# B&R Automation Studio project CControl_Gschneitner (part 7)

```iecst
		//Box 2 im Intervallbetrieb -> Dauerbetrieb u. Intervallbetrieb-Zeitfenster für alle anderen Boxen mit gleichem Lüfter sperren
		IF Box2In.IntervallbetriebEin THEN
			IF (Box2In.Ventilator1 AND Box1In.Ventilator1) OR (Box2In.Ventilator2 AND Box1In.Ventilator2) THEN
				Box1Out.DauerbetriebSperre	:= TRUE;
				FOR i := 0 TO 23 DO
					IF (Box2In.IntervallbetriebZeiten[i] = TRUE) THEN
						Box1Out.IntervallbetriebZeitenGesperrt[i]	:= TRUE;
					END_IF
				END_FOR
			END_IF
			IF (Box2In.Ventilator1 AND Box3In.Ventilator1) OR (Box2In.Ventilator2 AND Box3In.Ventilator2) THEN
				Box3Out.DauerbetriebSperre	:= TRUE;
				FOR i := 0 TO 23 DO
					IF (Box2In.IntervallbetriebZeiten[i] = TRUE) THEN
						Box3Out.IntervallbetriebZeitenGesperrt[i]	:= TRUE;
					END_IF
				END_FOR
			END_IF
			IF (Box2In.Ventilator1 AND Box4In.Ventilator1) OR (Box2In.Ventilator2 AND Box4In.Ventilator2) THEN
				Box4Out.DauerbetriebSperre	:= TRUE;
				FOR i := 0 TO 23 DO
					IF (Box2In.IntervallbetriebZeiten[i] = TRUE) THEN
						Box4Out.IntervallbetriebZeitenGesperrt[i]	:= TRUE;
					END_IF
				END_FOR
			END_IF
			IF (Box2In.Ventilator1 AND Box5In.Ventilator1) OR (Box2In.Ventilator2 AND Box5In.Ventilator2) THEN
				Box5Out.DauerbetriebSperre	:= TRUE;
				FOR i := 0 TO 23 DO
					IF (Box2In.IntervallbetriebZeiten[i] = TRUE) THEN
						Box5Out.IntervallbetriebZeitenGesperrt[i]	:= TRUE;
					END_IF
				END_FOR
			END_IF
			IF (Box2In.Ventilator1 AND Box6In.Ventilator1) OR (Box2In.Ventilator2 AND Box6In.Ventilator2) THEN
				Box6Out.DauerbetriebSperre	:= TRUE;
				FOR i := 0 TO 23 DO
					IF (Box2In.IntervallbetriebZeiten[i] = TRUE) THEN
						Box6Out.IntervallbetriebZeitenGesperrt[i]	:= TRUE;
					END_IF
				END_FOR
			END_IF
		END_IF

		//Box 3 im Intervallbetrieb -> Dauerbetrieb u. Intervallbetrieb-Zeitfenster für alle anderen Boxen mit gleichem Lüfter sperren
		IF Box3In.IntervallbetriebEin THEN
			IF (Box3In.Ventilator1 AND Box1In.Ventilator1) OR (Box3In.Ventilator2 AND Box1In.Ventilator2) THEN
				Box1Out.DauerbetriebSperre	:= TRUE;
				FOR i := 0 TO 23 DO
					IF (Box3In.IntervallbetriebZeiten[i] = TRUE) THEN
						Box1Out.IntervallbetriebZeitenGesperrt[i]	:= TRUE;
					END_IF
				END_FOR
			END_IF
			IF (Box3In.Ventilator1 AND Box2In.Ventilator1) OR (Box3In.Ventilator2 AND Box2In.Ventilator2) THEN
				Box2Out.DauerbetriebSperre	:= TRUE;
				FOR i := 0 TO 23 DO
					IF (Box3In.IntervallbetriebZeiten[i] = TRUE) THEN
						Box2Out.IntervallbetriebZeitenGesperrt[i]	:= TRUE;
					END_IF
				END_FOR
			END_IF
			IF (Box3In.Ventilator1 AND Box4In.Ventilator1) OR (Box3In.Ventilator2 AND Box4In.Ventilator2) THEN
				Box4Out.DauerbetriebSperre	:= TRUE;
				FOR i := 0 TO 23 DO
					IF (Box3In.IntervallbetriebZeiten[i] = TRUE) THEN
						Box4Out.IntervallbetriebZeitenGesperrt[i]	:= TRUE;
					END_IF
				END_FOR
			END_IF
			IF (Box3In.Ventilator1 AND Box5In.Ventilator1) OR (Box3In.Ventilator2 AND Box5In.Ventilator2) THEN
				Box5Out.DauerbetriebSperre	:= TRUE;
				FOR i := 0 TO 23 DO
					IF (Box3In.IntervallbetriebZeiten[i] = TRUE) THEN
						Box5Out.IntervallbetriebZeitenGesperrt[i]	:= TRUE;
					END_IF
				END_FOR
			END_IF
			IF (Box3In.Ventilator1 AND Box6In.Ventilator1) OR (Box3In.Ventilator2 AND Box6In.Ventilator2) THEN
				Box6Out.DauerbetriebSperre	:= TRUE;
				FOR i := 0 TO 23 DO
					IF (Box3In.IntervallbetriebZeiten[i] = TRUE) THEN
						Box6Out.IntervallbetriebZeitenGesperrt[i]	:= TRUE;
					END_IF
				END_FOR
			END_IF
		END_IF

		//Box 4 im Intervallbetrieb -> Dauerbetrieb u. Intervallbetrieb-Zeitfenster für alle anderen Boxen mit gleichem Lüfter sperren
		IF Box4In.IntervallbetriebEin THEN
			IF (Box4In.Ventilator1 AND Box1In.Ventilator1) OR (Box4In.Ventilator2 AND Box1In.Ventilator2) THEN
				Box1Out.DauerbetriebSperre	:= TRUE;
				FOR i := 0 TO 23 DO
					IF (Box4In.IntervallbetriebZeiten[i] = TRUE) THEN
						Box1Out.IntervallbetriebZeitenGesperrt[i]	:= TRUE;
					END_IF
				END_FOR
			END_IF
			IF (Box4In.Ventilator1 AND Box2In.Ventilator1) OR (Box4In.Ventilator2 AND Box2In.Ventilator2) THEN
				Box2Out.DauerbetriebSperre	:= TRUE;
				FOR i := 0 TO 23 DO
					IF (Box4In.IntervallbetriebZeiten[i] = TRUE) THEN
						Box2Out.IntervallbetriebZeitenGesperrt[i]	:= TRUE;
					END_IF
				END_FOR
			END_IF
			IF (Box4In.Ventilator1 AND Box3In.Ventilator1) OR (Box4In.Ventilator2 AND Box3In.Ventilator2) THEN
				Box3Out.DauerbetriebSperre	:= TRUE;
				FOR i := 0 TO 23 DO
					IF (Box4In.IntervallbetriebZeiten[i] = TRUE) THEN
						Box3Out.IntervallbetriebZeitenGesperrt[i]	:= TRUE;
					END_IF
				END_FOR
			END_IF
			IF (Box4In.Ventilator1 AND Box5In.Ventilator1) OR (Box4In.Ventilator2 AND Box5In.Ventilator2) THEN
				Box5Out.DauerbetriebSperre	:= TRUE;
				FOR i := 0 TO 23 DO
					IF (Box4In.IntervallbetriebZeiten[i] = TRUE) THEN
						Box5Out.IntervallbetriebZeitenGesperrt[i]	:= TRUE;
					END_IF
				END_FOR
			END_IF
			IF (Box4In.Ventilator1 AND Box6In.Ventilator1) OR (Box4In.Ventilator2 AND Box6In.Ventilator2) THEN
				Box6Out.DauerbetriebSperre	:= TRUE;
				FOR i := 0 TO 23 DO
					IF (Box4In.IntervallbetriebZeiten[i] = TRUE) THEN
						Box6Out.IntervallbetriebZeitenGesperrt[i]	:= TRUE;
					END_IF
				END_FOR
			END_IF
		END_IF

		//Box 5 im Intervallbetrieb -> Dauerbetrieb u. Intervallbetrieb-Zeitfenster für alle anderen Boxen mit gleichem Lüfter sperren
		IF Box5In.IntervallbetriebEin THEN
			IF (Box5In.Ventilator1 AND Box1In.Ventilator1) OR (Box5In.Ventilator2 AND Box1In.Ventilator2) THEN
				Box1Out.DauerbetriebSperre	:= TRUE;
				FOR i := 0 TO 23 DO
					IF (Box5In.IntervallbetriebZeiten[i] = TRUE) THEN
						Box1Out.IntervallbetriebZeitenGesperrt[i]	:= TRUE;
					END_IF
				END_FOR
			END_IF
			IF (Box5In.Ventilator1 AND Box2In.Ventilator1) OR (Box5In.Ventilator2 AND Box2In.Ventilator2) THEN
				Box2Out.DauerbetriebSperre	:= TRUE;
				FOR i := 0 TO 23 DO
					IF (Box5In.IntervallbetriebZeiten[i] = TRUE) THEN
						Box2Out.IntervallbetriebZeitenGesperrt[i]	:= TRUE;
					END_IF
				END_FOR
			END_IF
			IF (Box5In.Ventilator1 AND Box3In.Ventilator1) OR (Box5In.Ventilator2 AND Box3In.Ventilator2) THEN
				Box3Out.DauerbetriebSperre	:= TRUE;
				FOR i := 0 TO 23 DO
					IF (Box5In.IntervallbetriebZeiten[i] = TRUE) THEN
						Box3Out.IntervallbetriebZeitenGesperrt[i]	:= TRUE;
					END_IF
				END_FOR
			END_IF
			IF (Box5In.Ventilator1 AND Box4In.Ventilator1) OR (Box5In.Ventilator2 AND Box4In.Ventilator2) THEN
				Box4Out.DauerbetriebSperre	:= TRUE;
				FOR i := 0 TO 23 DO
					IF (Box5In.IntervallbetriebZeiten[i] = TRUE) THEN
						Box4Out.IntervallbetriebZeitenGesperrt[i]	:= TRUE;
					END_IF
				END_FOR
			END_IF
			IF (Box5In.Ventilator1 AND Box6In.Ventilator1) OR (Box5In.Ventilator2 AND Box6In.Ventilator2) THEN
				Box6Out.DauerbetriebSperre	:= TRUE;
				FOR i := 0 TO 23 DO
					IF (Box5In.IntervallbetriebZeiten[i] = TRUE) THEN
						Box6Out.IntervallbetriebZeitenGesperrt[i]	:= TRUE;
					END_IF
				END_FOR
			END_IF
		END_IF

		//Box 6 im Intervallbetrieb -> Dauerbetrieb u. Intervallbetrieb-Zeitfenster für alle anderen Boxen mit gleichem Lüfter sperren
		IF Box6In.IntervallbetriebEin THEN
			IF (Box6In.Ventilator1 AND Box1In.Ventilator1) OR (Box6In.Ventilator2 AND Box1In.Ventilator2) THEN
				Box1Out.DauerbetriebSperre	:= TRUE;
				FOR i := 0 TO 23 DO
					IF (Box6In.IntervallbetriebZeiten[i] = TRUE) THEN
						Box1Out.IntervallbetriebZeitenGesperrt[i]	:= TRUE;
					END_IF
				END_FOR
			END_IF
			IF (Box6In.Ventilator1 AND Box2In.Ventilator1) OR (Box6In.Ventilator2 AND Box2In.Ventilator2) THEN
				Box2Out.DauerbetriebSperre	:= TRUE;
				FOR i := 0 TO 23 DO
					IF (Box6In.IntervallbetriebZeiten[i] = TRUE) THEN
						Box2Out.IntervallbetriebZeitenGesperrt[i]	:= TRUE;
					END_IF
				END_FOR
			END_IF
			IF (Box6In.Ventilator1 AND Box3In.Ventilator1) OR (Box6In.Ventilator2 AND Box3In.Ventilator2) THEN
				Box3Out.DauerbetriebSperre	:= TRUE;
				FOR i := 0 TO 23 DO
					IF (Box6In.IntervallbetriebZeiten[i] = TRUE) THEN
						Box3Out.IntervallbetriebZeitenGesperrt[i]	:= TRUE;
					END_IF
				END_FOR
			END_IF
			IF (Box6In.Ventilator1 AND Box4In.Ventilator1) OR (Box6In.Ventilator2 AND Box4In.Ventilator2) THEN
				Box4Out.DauerbetriebSperre	:= TRUE;
				FOR i := 0 TO 23 DO
					IF (Box6In.IntervallbetriebZeiten[i] = TRUE) THEN
						Box4Out.IntervallbetriebZeitenGesperrt[i]	:= TRUE;
					END_IF
				END_FOR
			END_IF
			IF (Box6In.Ventilator1 AND Box5In.Ventilator1) OR (Box6In.Ventilator2 AND Box5In.Ventilator2) THEN
				Box5Out.DauerbetriebSperre	:= TRUE;
				FOR i := 0 TO 23 DO
					IF (Box6In.IntervallbetriebZeiten[i] = TRUE) THEN
						Box5Out.IntervallbetriebZeitenGesperrt[i]	:= TRUE;
					END_IF
				END_FOR
			END_IF
		END_IF

		//NACHTROCKNUNG AKTIVIERT =========================================================================================================================================================

		//Box 1 in der Nachtrocknung -> Nachtrocknungs-Zeitfenster für alle anderen Boxen mit gleichem Lüfter sperren
		IF Box1In.NachtrocknungEin THEN
			IF (Box1In.Ventilator1 AND Box2In.Ventilator1) OR (Box1In.Ventilator2 AND Box2In.Ventilator2) THEN
				FOR i := 0 TO 23 DO
					IF (Box1In.NachtrocknungZeiten[i] = TRUE) THEN
						Box2Out.NachtrocknungZeitenGesperrt[i]	:= TRUE;
					END_IF
				END_FOR
			END_IF
			IF (Box1In.Ventilator1 AND Box3In.Ventilator1) OR (Box1In.Ventilator2 AND Box3In.Ventilator2) THEN
				FOR i := 0 TO 23 DO
					IF (Box1In.NachtrocknungZeiten[i] = TRUE) THEN
						Box3Out.NachtrocknungZeitenGesperrt[i]	:= TRUE;
					END_IF
				END_FOR
			END_IF
			IF (Box1In.Ventilator1 AND Box4In.Ventilator1) OR (Box1In.Ventilator2 AND Box4In.Ventilator2) THEN
				FOR i := 0 TO 23 DO
					IF (Box1In.NachtrocknungZeiten[i] = TRUE) THEN
						Box4Out.NachtrocknungZeitenGesperrt[i]	:= TRUE;
					END_IF
				END_FOR
			END_IF
			IF (Box1In.Ventilator1 AND Box5In.Ventilator1) OR (Box1In.Ventilator2 AND Box5In.Ventilator2) THEN
				FOR i := 0 TO 23 DO
					IF (Box1In.NachtrocknungZeiten[i] = TRUE) THEN
						Box5Out.NachtrocknungZeitenGesperrt[i]	:= TRUE;
					END_IF
				END_FOR
			END_IF
			IF (Box1In.Ventilator1 AND Box6In.Ventilator1) OR (Box1In.Ventilator2 AND Box6In.Ventilator2) THEN
				FOR i := 0 TO 23 DO
					IF (Box1In.NachtrocknungZeiten[i] = TRUE) THEN
						Box6Out.NachtrocknungZeitenGesperrt[i]	:= TRUE;
					END_IF
				END_FOR
			END_IF
		END_IF

		//Box 2 in der Nachtrocknung -> Nachtrocknungs-Zeitfenster für alle anderen Boxen mit gleichem Lüfter sperren
		IF Box2In.NachtrocknungEin THEN
			IF (Box2In.Ventilator1 AND Box1In.Ventilator1) OR (Box2In.Ventilator2 AND Box1In.Ventilator2) THEN
				FOR i := 0 TO 23 DO
					IF (Box2In.NachtrocknungZeiten[i] = TRUE) THEN
						Box1Out.NachtrocknungZeitenGesperrt[i]	:= TRUE;
					END_IF
				END_FOR
			END_IF
			IF (Box2In.Ventilator1 AND Box3In.Ventilator1) OR (Box2In.Ventilator2 AND Box3In.Ventilator2) THEN
				FOR i := 0 TO 23 DO
					IF (Box2In.NachtrocknungZeiten[i] = TRUE) THEN
						Box3Out.NachtrocknungZeitenGesperrt[i]	:= TRUE;
					END_IF
				END_FOR
			END_IF
			IF (Box2In.Ventilator1 AND Box4In.Ventilator1) OR (Box2In.Ventilator2 AND Box4In.Ventilator2) THEN
				FOR i := 0 TO 23 DO
					IF (Box2In.NachtrocknungZeiten[i] = TRUE) THEN
						Box4Out.NachtrocknungZeitenGesperrt[i]	:= TRUE;
					END_IF
				END_FOR
			END_IF
			IF (Box2In.Ventilator1 AND Box5In.Ventilator1) OR (Box2In.Ventilator2 AND Box5In.Ventilator2) THEN
				FOR i := 0 TO 23 DO
					IF (Box2In.NachtrocknungZeiten[i] = TRUE) THEN
						Box5Out.NachtrocknungZeitenGesperrt[i]	:= TRUE;
					END_IF
				END_FOR
			END_IF
			IF (Box2In.Ventilator1 AND Box6In.Ventilator1) OR (Box2In.Ventilator2 AND Box6In.Ventilator2) THEN
				FOR i := 0 TO 23 DO
					IF (Box2In.NachtrocknungZeiten[i] = TRUE) THEN
						Box6Out.NachtrocknungZeitenGesperrt[i]	:= TRUE;
					END_IF
				END_FOR
			END_IF
		END_IF

		//Box 3 in der Nachtrocknung -> Nachtrocknungs-Zeitfenster für alle anderen Boxen mit gleichem Lüfter sperren
		IF Box3In.NachtrocknungEin THEN
			IF (Box3In.Ventilator1 AND Box1In.Ventilator1) OR (Box3In.Ventilator2 AND Box1In.Ventilator2) THEN
				FOR i := 0 TO 23 DO
					IF (Box3In.NachtrocknungZeiten[i] = TRUE) THEN
						Box1Out.NachtrocknungZeitenGesperrt[i]	:= TRUE;
					END_IF
				END_FOR
			END_IF
			IF (Box3In.Ventilator1 AND Box2In.Ventilator1) OR (Box3In.Ventilator2 AND Box2In.Ventilator2) THEN
				FOR i := 0 TO 23 DO
					IF (Box3In.NachtrocknungZeiten[i] = TRUE) THEN
						Box2Out.NachtrocknungZeitenGesperrt[i]	:= TRUE;
					END_IF
				END_FOR
			END_IF
			IF (Box3In.Ventilator1 AND Box4In.Ventilator1) OR (Box3In.Ventilator2 AND Box4In.Ventilator2) THEN
				FOR i := 0 TO 23 DO
					IF (Box3In.NachtrocknungZeiten[i] = TRUE) THEN
						Box4Out.NachtrocknungZeitenGesperrt[i]	:= TRUE;
					END_IF
				END_FOR
			END_IF
			IF (Box3In.Ventilator1 AND Box5In.Ventilator1) OR (Box3In.Ventilator2 AND Box5In.Ventilator2) THEN
				FOR i := 0 TO 23 DO
					IF (Box3In.NachtrocknungZeiten[i] = TRUE) THEN
						Box5Out.NachtrocknungZeitenGesperrt[i]	:= TRUE;
					END_IF
				END_FOR
			END_IF
			IF (Box3In.Ventilator1 AND Box6In.Ventilator1) OR (Box3In.Ventilator2 AND Box6In.Ventilator2) THEN
				FOR i := 0 TO 23 DO
					IF (Box3In.NachtrocknungZeiten[i] = TRUE) THEN
						Box6Out.NachtrocknungZeitenGesperrt[i]	:= TRUE;
					END_IF
				END_FOR
			END_IF
		END_IF

		//Box 4 in der Nachtrocknung -> Nachtrocknungs-Zeitfenster für alle anderen Boxen mit gleichem Lüfter sperren
		IF Box4In.NachtrocknungEin THEN
			IF (Box4In.Ventilator1 AND Box1In.Ventilator1) OR (Box4In.Ventilator2 AND Box1In.Ventilator2) THEN
				FOR i := 0 TO 23 DO
					IF (Box4In.NachtrocknungZeiten[i] = TRUE) THEN
						Box1Out.NachtrocknungZeitenGesperrt[i]	:= TRUE;
					END_IF
				END_FOR
			END_IF
			IF (Box4In.Ventilator1 AND Box2In.Ventilator1) OR (Box4In.Ventilator2 AND Box2In.Ventilator2) THEN
				FOR i := 0 TO 23 DO
					IF (Box4In.NachtrocknungZeiten[i] = TRUE) THEN
						Box2Out.NachtrocknungZeitenGesperrt[i]	:= TRUE;
					END_IF
				END_FOR
			END_IF
			IF (Box4In.Ventilator1 AND Box3In.Ventilator1) OR (Box4In.Ventilator2 AND Box3In.Ventilator2) THEN
				FOR i := 0 TO 23 DO
					IF (Box4In.NachtrocknungZeiten[i] = TRUE) THEN
						Box3Out.NachtrocknungZeitenGesperrt[i]	:= TRUE;
					END_IF
				END_FOR
			END_IF
			IF (Box4In.Ventilator1 AND Box5In.Ventilator1) OR (Box4In.Ventilator2 AND Box5In.Ventilator2) THEN
				FOR i := 0 TO 23 DO
					IF (Box4In.NachtrocknungZeiten[i] = TRUE) THEN
						Box5Out.NachtrocknungZeitenGesperrt[i]	:= TRUE;
					END_IF
				END_FOR
			END_IF
			IF (Box4In.Ventilator1 AND Box6In.Ventilator1) OR (Box4In.Ventilator2 AND Box6In.Ventilator2) THEN
				FOR i := 0 TO 23 DO
					IF (Box4In.NachtrocknungZeiten[i] = TRUE) THEN
						Box6Out.NachtrocknungZeitenGesperrt[i]	:= TRUE;
					END_IF
				END_FOR
			END_IF
		END_IF

		//Box 5 in der Nachtrocknung -> Nachtrocknungs-Zeitfenster für alle anderen Boxen mit gleichem Lüfter sperren
		IF Box5In.NachtrocknungEin THEN
			IF (Box5In.Ventilator1 AND Box1In.Ventilator1) OR (Box5In.Ventilator2 AND Box1In.Ventilator2) THEN
				FOR i := 0 TO 23 DO
					IF (Box5In.NachtrocknungZeiten[i] = TRUE) THEN
						Box1Out.NachtrocknungZeitenGesperrt[i]	:= TRUE;
					END_IF
				END_FOR
			END_IF
			IF (Box5In.Ventilator1 AND Box2In.Ventilator1) OR (Box5In.Ventilator2 AND Box2In.Ventilator2) THEN
				FOR i := 0 TO 23 DO
					IF (Box5In.NachtrocknungZeiten[i] = TRUE) THEN
						Box2Out.NachtrocknungZeitenGesperrt[i]	:= TRUE;
					END_IF
				END_FOR
			END_IF
			IF (Box5In.Ventilator1 AND Box3In.Ventilator1) OR (Box5In.Ventilator2 AND Box3In.Ventilator2) THEN
				FOR i := 0 TO 23 DO
					IF (Box5In.NachtrocknungZeiten[i] = TRUE) THEN
						Box3Out.NachtrocknungZeitenGesperrt[i]	:= TRUE;
					END_IF
				END_FOR
			END_IF
			IF (Box5In.Ventilator1 AND Box4In.Ventilator1) OR (Box5In.Ventilator2 AND Box4In.Ventilator2) THEN
				FOR i := 0 TO 23 DO
					IF (Box5In.NachtrocknungZeiten[i] = TRUE) THEN
						Box4Out.NachtrocknungZeitenGesperrt[i]	:= TRUE;
					END_IF
				END_FOR
			END_IF
			IF (Box5In.Ventilator1 AND Box6In.Ventilator1) OR (Box5In.Ventilator2 AND Box6In.Ventilator2) THEN
				FOR i := 0 TO 23 DO
					IF (Box5In.NachtrocknungZeiten[i] = TRUE) THEN
						Box6Out.NachtrocknungZeitenGesperrt[i]	:= TRUE;
					END_IF
				END_FOR
			END_IF
		END_IF

		//Box 6 in der Nachtrocknung -> Nachtrocknungs-Zeitfenster für alle anderen Boxen mit gleichem Lüfter sperren
		IF Box6In.NachtrocknungEin THEN
			IF (Box6In.Ventilator1 AND Box1In.Ventilator1) OR (Box6In.Ventilator2 AND Box1In.Ventilator2) THEN
				FOR i := 0 TO 23 DO
					IF (Box6In.NachtrocknungZeiten[i] = TRUE) THEN
						Box1Out.NachtrocknungZeitenGesperrt[i]	:= TRUE;
					END_IF
				END_FOR
			END_IF
			IF (Box6In.Ventilator1 AND Box2In.Ventilator1) OR (Box6In.Ventilator2 AND Box2In.Ventilator2) THEN
				FOR i := 0 TO 23 DO
					IF (Box6In.NachtrocknungZeiten[i] = TRUE) THEN
						Box2Out.NachtrocknungZeitenGesperrt[i]	:= TRUE;
					END_IF
				END_FOR
			END_IF
			IF (Box6In.Ventilator1 AND Box3In.Ventilator1) OR (Box6In.Ventilator2 AND Box3In.Ventilator2) THEN
				FOR i := 0 TO 23 DO
					IF (Box6In.NachtrocknungZeiten[i] = TRUE) THEN
						Box3Out.NachtrocknungZeitenGesperrt[i]	:= TRUE;
					END_IF
				END_FOR
			END_IF
			IF (Box6In.Ventilator1 AND Box4In.Ventilator1) OR (Box6In.Ventilator2 AND Box4In.Ventilator2) THEN
				FOR i := 0 TO 23 DO
					IF (Box6In.NachtrocknungZeiten[i] = TRUE) THEN
						Box4Out.NachtrocknungZeitenGesperrt[i]	:= TRUE;
					END_IF
				END_FOR
			END_IF
			IF (Box6In.Ventilator1 AND Box5In.Ventilator1) OR (Box6In.Ventilator2 AND Box5In.Ventilator2) THEN
				FOR i := 0 TO 23 DO
					IF (Box6In.NachtrocknungZeiten[i] = TRUE) THEN
						Box5Out.NachtrocknungZeitenGesperrt[i]	:= TRUE;
					END_IF
				END_FOR
			END_IF
		END_IF

		//Mehrere Boxen gleichzeitig belüftbar (Jalousieklappen) ******************************************************************************************************************
	ELSE

		//Box 1
		Box1Out.DauerbetriebSperre		:= FALSE;
		Box1Out.IntervallbetriebSperre	:= FALSE;
		memset(ADR(Box1Out.IntervallbetriebZeitenGesperrt), 0, SIZEOF(Box1Out.IntervallbetriebZeitenGesperrt));
		memset(ADR(Box1Out.NachtrocknungZeitenGesperrt), 0, SIZEOF(Box1Out.NachtrocknungZeitenGesperrt));

		//Box 2
		Box2Out.DauerbetriebSperre		:= FALSE;
		Box2Out.IntervallbetriebSperre	:= FALSE;
		memset(ADR(Box2Out.IntervallbetriebZeitenGesperrt), 0, SIZEOF(Box2Out.IntervallbetriebZeitenGesperrt));
		memset(ADR(Box2Out.NachtrocknungZeitenGesperrt), 0, SIZEOF(Box2Out.NachtrocknungZeitenGesperrt));

		//Box 3
		Box3Out.DauerbetriebSperre		:= FALSE;
		Box3Out.IntervallbetriebSperre	:= FALSE;
		memset(ADR(Box3Out.IntervallbetriebZeitenGesperrt), 0, SIZEOF(Box3Out.IntervallbetriebZeitenGesperrt));
		memset(ADR(Box3Out.NachtrocknungZeitenGesperrt), 0, SIZEOF(Box3Out.NachtrocknungZeitenGesperrt));

		//Box 4
		Box4Out.DauerbetriebSperre		:= FALSE;
		Box4Out.IntervallbetriebSperre	:= FALSE;
		memset(ADR(Box4Out.IntervallbetriebZeitenGesperrt), 0, SIZEOF(Box4Out.IntervallbetriebZeitenGesperrt));
		memset(ADR(Box4Out.NachtrocknungZeitenGesperrt), 0, SIZEOF(Box4Out.NachtrocknungZeitenGesperrt));

		//Box 5
		Box5Out.DauerbetriebSperre		:= FALSE;
		Box5Out.IntervallbetriebSperre	:= FALSE;
		memset(ADR(Box5Out.IntervallbetriebZeitenGesperrt), 0, SIZEOF(Box5Out.IntervallbetriebZeitenGesperrt));
		memset(ADR(Box5Out.NachtrocknungZeitenGesperrt), 0, SIZEOF(Box5Out.NachtrocknungZeitenGesperrt));

		//Box 6
		Box6Out.DauerbetriebSperre		:= FALSE;
		Box6Out.IntervallbetriebSperre	:= FALSE;
		memset(ADR(Box6Out.IntervallbetriebZeitenGesperrt), 0, SIZEOF(Box6Out.IntervallbetriebZeitenGesperrt));
		memset(ADR(Box6Out.NachtrocknungZeitenGesperrt), 0, SIZEOF(Box6Out.NachtrocknungZeitenGesperrt));

	END_IF

	//===================================================================================================================================================================================================
	//Abhängigkeiten der Boxenklappen und Bypassklappe zu den Ventilatoren ermitteln
	//(damit bei Klappenumschaltung Anlagen mit 2 Ventilatoren nur der zuständige Ventilator abgeschaltet wird)
	//===================================================================================================================================================================================================

	//Boxenklappe 1 - Ventilator 1
	Boxenkl1VonVent1Abhaengig := (Box1In.Ventilator1 AND (Box1In.StellungKlappe1 <> FBBOX_NICHT_VERWENDET)) OR
	(Box2In.Ventilator1 AND (Box2In.StellungKlappe1 <> FBBOX_NICHT_VERWENDET)) OR (Box3In.Ventilator1 AND (Box3In.StellungKlappe1 <> FBBOX_NICHT_VERWENDET)) OR
	(Box4In.Ventilator1 AND (Box4In.StellungKlappe1 <> FBBOX_NICHT_VERWENDET)) OR (Box5In.Ventilator1 AND (Box5In.StellungKlappe1 <> FBBOX_NICHT_VERWENDET)) OR
	(Box6In.Ventilator1 AND (Box6In.StellungKlappe1 <> FBBOX_NICHT_VERWENDET)) OR BoxenklVonBeidenVentAbhaengig;

	//Boxenklappe 1 - Ventilator 2
	Boxenkl1VonVent2Abhaengig := (Box1In.Ventilator2 AND (Box1In.StellungKlappe1 <> FBBOX_NICHT_VERWENDET)) OR
	(Box2In.Ventilator2 AND (Box2In.StellungKlappe1 <> FBBOX_NICHT_VERWENDET)) OR (Box3In.Ventilator2 AND (Box3In.StellungKlappe1 <> FBBOX_NICHT_VERWENDET)) OR
	(Box4In.Ventilator2 AND (Box4In.StellungKlappe1 <> FBBOX_NICHT_VERWENDET)) OR (Box5In.Ventilator2 AND (Box5In.StellungKlappe1 <> FBBOX_NICHT_VERWENDET)) OR
	(Box6In.Ventilator2 AND (Box6In.StellungKlappe1 <> FBBOX_NICHT_VERWENDET)) OR BoxenklVonBeidenVentAbhaengig;

	//Boxenklappe 2 - Ventilator 1
	Boxenkl2VonVent1Abhaengig := (Box1In.Ventilator1 AND (Box1In.StellungKlappe2 <> FBBOX_NICHT_VERWENDET)) OR
	(Box2In.Ventilator1 AND (Box2In.StellungKlappe2 <> FBBOX_NICHT_VERWENDET)) OR (Box3In.Ventilator1 AND (Box3In.StellungKlappe2 <> FBBOX_NICHT_VERWENDET)) OR
	(Box4In.Ventilator1 AND (Box4In.StellungKlappe2 <> FBBOX_NICHT_VERWENDET)) OR (Box5In.Ventilator1 AND (Box5In.StellungKlappe2 <> FBBOX_NICHT_VERWENDET)) OR
	(Box6In.Ventilator1 AND (Box6In.StellungKlappe2 <> FBBOX_NICHT_VERWENDET)) OR BoxenklVonBeidenVentAbhaengig;

	//Boxenklappe 2 - Ventilator 2
	Boxenkl2VonVent2Abhaengig := (Box1In.Ventilator2 AND (Box1In.StellungKlappe2 <> FBBOX_NICHT_VERWENDET)) OR
	(Box2In.Ventilator2 AND (Box2In.StellungKlappe2 <> FBBOX_NICHT_VERWENDET)) OR (Box3In.Ventilator2 AND (Box3In.StellungKlappe2 <> FBBOX_NICHT_VERWENDET)) OR
	(Box4In.Ventilator2 AND (Box4In.StellungKlappe2 <> FBBOX_NICHT_VERWENDET)) OR (Box5In.Ventilator2 AND (Box5In.StellungKlappe2 <> FBBOX_NICHT_VERWENDET)) OR
	(Box6In.Ventilator2 AND (Box6In.StellungKlappe2 <> FBBOX_NICHT_VERWENDET)) OR BoxenklVonBeidenVentAbhaengig;

	//Boxenklappe 3 - Ventilator 1
	Boxenkl3VonVent1Abhaengig := (Box1In.Ventilator1 AND (Box1In.StellungKlappe3 <> FBBOX_NICHT_VERWENDET)) OR
	(Box2In.Ventilator1 AND (Box2In.StellungKlappe3 <> FBBOX_NICHT_VERWENDET)) OR (Box3In.Ventilator1 AND (Box3In.StellungKlappe3 <> FBBOX_NICHT_VERWENDET)) OR
	(Box4In.Ventilator1 AND (Box4In.StellungKlappe3 <> FBBOX_NICHT_VERWENDET)) OR (Box5In.Ventilator1 AND (Box5In.StellungKlappe3 <> FBBOX_NICHT_VERWENDET)) OR
	(Box6In.Ventilator1 AND (Box6In.StellungKlappe3 <> FBBOX_NICHT_VERWENDET)) OR BoxenklVonBeidenVentAbhaengig;

	//Boxenklappe 3 - Ventilator 2
	Boxenkl3VonVent2Abhaengig := (Box1In.Ventilator2 AND (Box1In.StellungKlappe3 <> FBBOX_NICHT_VERWENDET)) OR
	(Box2In.Ventilator2 AND (Box2In.StellungKlappe3 <> FBBOX_NICHT_VERWENDET)) OR (Box3In.Ventilator2 AND (Box3In.StellungKlappe3 <> FBBOX_NICHT_VERWENDET)) OR
	(Box4In.Ventilator2 AND (Box4In.StellungKlappe3 <> FBBOX_NICHT_VERWENDET)) OR (Box5In.Ventilator2 AND (Box5In.StellungKlappe3 <> FBBOX_NICHT_VERWENDET)) OR
	(Box6In.Ventilator2 AND (Box6In.StellungKlappe3 <> FBBOX_NICHT_VERWENDET)) OR BoxenklVonBeidenVentAbhaengig;

	//Boxenklappe 4 - Ventilator 1
	Boxenkl4VonVent1Abhaengig := (Box1In.Ventilator1 AND (Box1In.StellungKlappe4 <> FBBOX_NICHT_VERWENDET)) OR
	(Box2In.Ventilator1 AND (Box2In.StellungKlappe4 <> FBBOX_NICHT_VERWENDET)) OR (Box3In.Ventilator1 AND (Box3In.StellungKlappe4 <> FBBOX_NICHT_VERWENDET)) OR
	(Box4In.Ventilator1 AND (Box4In.StellungKlappe4 <> FBBOX_NICHT_VERWENDET)) OR (Box5In.Ventilator1 AND (Box5In.StellungKlappe4 <> FBBOX_NICHT_VERWENDET)) OR
	(Box6In.Ventilator1 AND (Box6In.StellungKlappe4 <> FBBOX_NICHT_VERWENDET)) OR BoxenklVonBeidenVentAbhaengig;

	//Boxenklappe 4 - Ventilator 2
	Boxenkl4VonVent2Abhaengig := (Box1In.Ventilator2 AND (Box1In.StellungKlappe4 <> FBBOX_NICHT_VERWENDET)) OR
	(Box2In.Ventilator2 AND (Box2In.StellungKlappe4 <> FBBOX_NICHT_VERWENDET)) OR (Box3In.Ventilator2 AND (Box3In.StellungKlappe4 <> FBBOX_NICHT_VERWENDET)) OR
	(Box4In.Ventilator2 AND (Box4In.StellungKlappe4 <> FBBOX_NICHT_VERWENDET)) OR (Box5In.Ventilator2 AND (Box5In.StellungKlappe4 <> FBBOX_NICHT_VERWENDET)) OR
	(Box6In.Ventilator2 AND (Box6In.StellungKlappe4 <> FBBOX_NICHT_VERWENDET)) OR BoxenklVonBeidenVentAbhaengig;

	//Boxenklappe 5 - Ventilator 1
	Boxenkl5VonVent1Abhaengig := (Box1In.Ventilator1 AND (Box1In.StellungKlappe5 <> FBBOX_NICHT_VERWENDET)) OR
	(Box2In.Ventilator1 AND (Box2In.StellungKlappe5 <> FBBOX_NICHT_VERWENDET)) OR (Box3In.Ventilator1 AND (Box3In.StellungKlappe5 <> FBBOX_NICHT_VERWENDET)) OR
	(Box4In.Ventilator1 AND (Box4In.StellungKlappe5 <> FBBOX_NICHT_VERWENDET)) OR (Box5In.Ventilator1 AND (Box5In.StellungKlappe5 <> FBBOX_NICHT_VERWENDET)) OR
	(Box6In.Ventilator1 AND (Box6In.StellungKlappe5 <> FBBOX_NICHT_VERWENDET)) OR BoxenklVonBeidenVentAbhaengig;

	//Boxenklappe 5 - Ventilator 2
	Boxenkl5VonVent2Abhaengig := (Box1In.Ventilator2 AND (Box1In.StellungKlappe5 <> FBBOX_NICHT_VERWENDET)) OR
	(Box2In.Ventilator2 AND (Box2In.StellungKlappe5 <> FBBOX_NICHT_VERWENDET)) OR (Box3In.Ventilator2 AND (Box3In.StellungKlappe5 <> FBBOX_NICHT_VERWENDET)) OR
	(Box4In.Ventilator2 AND (Box4In.StellungKlappe5 <> FBBOX_NICHT_VERWENDET)) OR (Box5In.Ventilator2 AND (Box5In.StellungKlappe5 <> FBBOX_NICHT_VERWENDET)) OR
	(Box6In.Ventilator2 AND (Box6In.StellungKlappe5 <> FBBOX_NICHT_VERWENDET)) OR BoxenklVonBeidenVentAbhaengig;

	//Boxenklappe 6 - Ventilator 1
	Boxenkl6VonVent1Abhaengig := (Box1In.Ventilator1 AND (Box1In.StellungKlappe6 <> FBBOX_NICHT_VERWENDET)) OR
	(Box2In.Ventilator1 AND (Box2In.StellungKlappe6 <> FBBOX_NICHT_VERWENDET)) OR (Box3In.Ventilator1 AND (Box3In.StellungKlappe6 <> FBBOX_NICHT_VERWENDET)) OR
	(Box4In.Ventilator1 AND (Box4In.StellungKlappe6 <> FBBOX_NICHT_VERWENDET)) OR (Box5In.Ventilator1 AND (Box5In.StellungKlappe6 <> FBBOX_NICHT_VERWENDET)) OR
	(Box6In.Ventilator1 AND (Box6In.StellungKlappe6 <> FBBOX_NICHT_VERWENDET)) OR BoxenklVonBeidenVentAbhaengig;

	//Boxenklappe 6 - Ventilator 2
	Boxenkl6VonVent2Abhaengig := (Box1In.Ventilator2 AND (Box1In.StellungKlappe6 <> FBBOX_NICHT_VERWENDET)) OR
	(Box2In.Ventilator2 AND (Box2In.StellungKlappe6 <> FBBOX_NICHT_VERWENDET)) OR (Box3In.Ventilator2 AND (Box3In.StellungKlappe6 <> FBBOX_NICHT_VERWENDET)) OR
	(Box4In.Ventilator2 AND (Box4In.StellungKlappe6 <> FBBOX_NICHT_VERWENDET)) OR (Box5In.Ventilator2 AND (Box5In.StellungKlappe6 <> FBBOX_NICHT_VERWENDET)) OR
	(Box6In.Ventilator2 AND (Box6In.StellungKlappe6 <> FBBOX_NICHT_VERWENDET)) OR BoxenklVonBeidenVentAbhaengig;

	//Bypassklappe & Ventilator 1
	BypassklVonVent1Abhaengig := (Box1In.Ventilator1 AND Box1In.Luftentfeuchter) OR (Box2In.Ventilator1 AND Box2In.Luftentfeuchter) OR
	(Box3In.Ventilator1 AND Box3In.Luftentfeuchter) OR (Box4In.Ventilator1 AND Box4In.Luftentfeuchter) OR
	(Box5In.Ventilator1 AND Box5In.Luftentfeuchter) OR (Box6In.Ventilator1 AND Box6In.Luftentfeuchter) OR BypassklVonBeidenVentAbhaengig;

	//Bypassklappe & Ventilator 2
	BypassklVonVent2Abhaengig := (Box1In.Ventilator2 AND Box1In.Luftentfeuchter) OR (Box2In.Ventilator2 AND Box2In.Luftentfeuchter) OR
	(Box3In.Ventilator2 AND Box3In.Luftentfeuchter) OR (Box4In.Ventilator2 AND Box4In.Luftentfeuchter) OR
	(Box5In.Ventilator2 AND Box5In.Luftentfeuchter) OR (Box6In.Ventilator2 AND Box6In.Luftentfeuchter) OR BypassklVonBeidenVentAbhaengig;

END_FUNCTION_BLOCK
```

#### fbBoxenVentKlappen.st
```iecst
(* Funktionsbaustein für Ansteuerung Ventilatoren und Klappen *)
FUNCTION_BLOCK fbBoxenVentKlappen

	IF Freigabe THEN

		//Zeitticks erzeugen
		fbLascoEUhr_0(Freigabe := TRUE);
		fbLascoZdxx_0(IN := fbLascoEUhr_0.Sekunde);
		sekTick	:= fbLascoZdxx_0.Q;

		//Abfrage, ob Umschaltung Klappen erforderlich

		loc_AenderungBypassklappe		:= ((BypassklappeOeffnen AND NOT (EndlBypassOffen OR Bypassklappe.KlappeIstOffenOut)) OR
		(BypassklappeSchliessen AND NOT (EndlBypassGeschl OR Bypassklappe.KlappeIstGeschlOut))) AND (LaufzeitBypassklappe <> 0);

		loc_AenderungUmschaltklappe1	:= ((Umschaltkl1Oeffnen AND NOT (EndlUmschaltkl1Offen OR Umschaltklappe1.KlappeIstOffenOut)) OR
		(Umschaltkl1Schliessen AND NOT (EndlUmschaltkl1Geschl OR Umschaltklappe1.KlappeIstGeschlOut))) AND (LaufzeitUmschaltklappe1 <> 0);

		loc_AenderungUmschaltklappe2	:= ((Umschaltkl2Oeffnen AND NOT (EndlUmschaltkl2Offen OR Umschaltklappe2.KlappeIstOffenOut)) OR
		(Umschaltkl2Schliessen AND NOT (EndlUmschaltkl2Geschl OR Umschaltklappe2.KlappeIstGeschlOut))) AND (LaufzeitUmschaltklappe2 <> 0);

		loc_AenderungBoxenklappe1		:= Boxenklappe1Vorhanden AND ((Boxenklappe1Oeffnen AND NOT (EndlBoxenklappe1Offen OR Boxenklappe1.KlappeIstOffenOut)) OR
		(Boxenklappe1Schliessen AND NOT (EndlBoxenklappe1Geschl OR Boxenklappe1.KlappeIstGeschlOut))) AND (LaufzeitBoxenklappe1 <> 0);

		loc_AenderungBoxenklappe2		:= Boxenklappe2Vorhanden AND ((Boxenklappe2Oeffnen AND NOT (EndlBoxenklappe2Offen OR Boxenklappe2.KlappeIstOffenOut)) OR
		(Boxenklappe2Schliessen AND NOT (EndlBoxenklappe2Geschl OR Boxenklappe2.KlappeIstGeschlOut))) AND (LaufzeitBoxenklappe2 <> 0);

		loc_AenderungBoxenklappe3		:= Boxenklappe3Vorhanden AND ((Boxenklappe3Oeffnen AND NOT (EndlBoxenklappe3Offen OR Boxenklappe3.KlappeIstOffenOut)) OR
		(Boxenklappe3Schliessen AND NOT (EndlBoxenklappe3Geschl OR Boxenklappe3.KlappeIstGeschlOut))) AND (LaufzeitBoxenklappe3 <> 0);

		loc_AenderungBoxenklappe4		:= Boxenklappe4Vorhanden AND ((Boxenklappe4Oeffnen AND NOT (EndlBoxenklappe4Offen OR Boxenklappe4.KlappeIstOffenOut)) OR
		(Boxenklappe4Schliessen AND NOT (EndlBoxenklappe4Geschl OR Boxenklappe4.KlappeIstGeschlOut))) AND (LaufzeitBoxenklappe4 <> 0);

		loc_AenderungBoxenklappe5		:= Boxenklappe5Vorhanden AND ((Boxenklappe5Oeffnen AND NOT (EndlBoxenklappe5Offen OR Boxenklappe5.KlappeIstOffenOut)) OR
		(Boxenklappe5Schliessen AND NOT (EndlBoxenklappe5Geschl OR Boxenklappe5.KlappeIstGeschlOut))) AND (LaufzeitBoxenklappe5 <> 0);

		loc_AenderungBoxenklappe6		:= Boxenklappe6Vorhanden AND ((Boxenklappe6Oeffnen AND NOT (EndlBoxenklappe6Offen OR Boxenklappe6.KlappeIstOffenOut)) OR
		(Boxenklappe6Schliessen AND NOT (EndlBoxenklappe6Geschl OR Boxenklappe6.KlappeIstGeschlOut))) AND (LaufzeitBoxenklappe6 <> 0);

		//Umschaltung erforderlich bei Ventilator 1
		loc_UmschaltungErforderlVent1		:= (loc_AenderungBypassklappe AND BypassklVonVent1Abhaengig) OR
		(loc_AenderungUmschaltklappe1 AND UmluftklVonVent1Abhaengig) OR (loc_AenderungUmschaltklappe2 AND UmluftklVonVent1Abhaengig) OR
		(loc_AenderungBoxenklappe1 AND Boxenkl1VonVent1Abhaengig) OR (loc_AenderungBoxenklappe2 AND Boxenkl2VonVent1Abhaengig) OR
		(loc_AenderungBoxenklappe3 AND Boxenkl3VonVent1Abhaengig) OR (loc_AenderungBoxenklappe4 AND Boxenkl4VonVent1Abhaengig) OR
		(loc_AenderungBoxenklappe5 AND Boxenkl5VonVent1Abhaengig) OR (loc_AenderungBoxenklappe6 AND Boxenkl6VonVent1Abhaengig);

		//Umschaltung erfoderlich bei Ventilator 2
		loc_UmschaltungErforderlVent2		:= (loc_AenderungBypassklappe AND BypassklVonVent2Abhaengig) OR
		(loc_AenderungUmschaltklappe1 AND UmluftklVonVent2Abhaengig) OR (loc_AenderungUmschaltklappe2 AND UmluftklVonVent2Abhaengig) OR
		(loc_AenderungBoxenklappe1 AND Boxenkl1VonVent2Abhaengig) OR (loc_AenderungBoxenklappe2 AND Boxenkl2VonVent2Abhaengig) OR
		(loc_AenderungBoxenklappe3 AND Boxenkl3VonVent2Abhaengig) OR (loc_AenderungBoxenklappe4 AND Boxenkl4VonVent2Abhaengig) OR
		(loc_AenderungBoxenklappe5 AND Boxenkl5VonVent2Abhaengig) OR (loc_AenderungBoxenklappe6 AND Boxenkl6VonVent2Abhaengig);

		//Funktionsbaustein Ansteuerung FU Ventilator 1
		fbFuVentilator1.AnsprechZeitFU		:= 5;
		fbFuVentilator1.BetrMldg			:= Ventilator1InBetrieb;
		fbFuVentilator1.MinDrehzahl			:= DrehzahlVent1Min;
		fbFuVentilator1.MaxDrehzahl			:= DrehzahlVent1Max;
		fbFuVentilator1.RampeUpSek			:= RampeVent1Up;
		fbFuVentilator1.RampeDownSek		:= RampeVent1Down;
		fbFuVentilator1.Reset				:= QuitFehler;
		fbFuVentilator1.Tick				:= sekTick;
		fbFuVentilator1();
		FreigabeVentilator1Out				:= fbFuVentilator1.BetriebFU;
		DrehzahlVent1Out					:= fbFuVentilator1.DrehzahlFU;
		FehlerFuVentilator1					:= fbFuVentilator1.StoerungFU;

		//Funktionsbaustein Ansteuerung FU Ventilator 2
		fbFuVentilator2.AnsprechZeitFU		:= 5;
		fbFuVentilator2.BetrMldg			:= Ventilator2InBetrieb;
		fbFuVentilator2.MinDrehzahl			:= DrehzahlVent2Min;
		fbFuVentilator2.MaxDrehzahl			:= DrehzahlVent2Max;
		fbFuVentilator2.RampeUpSek			:= RampeVent2Up;
		fbFuVentilator2.RampeDownSek		:= RampeVent2Down;
		fbFuVentilator2.Reset				:= QuitFehler;
		fbFuVentilator2.Tick				:= sekTick;
		fbFuVentilator2();
		FreigabeVentilator2Out				:= fbFuVentilator2.BetriebFU;
		DrehzahlVent2Out					:= fbFuVentilator2.DrehzahlFU;
		FehlerFuVentilator2					:= fbFuVentilator2.StoerungFU;

		//Funktionsbausteine Klappen
		Bypassklappe.EndlagenVhd			:= EndlagenVhdBypassklappe;
		Bypassklappe.EndlageOffen			:= EndlBypassOffen;
		Bypassklappe.EndlageGeschl			:= EndlBypassGeschl;
		Bypassklappe.LaufzeitOeffnen		:= LaufzeitBypassklappe;
		Bypassklappe.LaufzeitSchliessen		:= LaufzeitBypassklappe;
		Bypassklappe.Stoerung				:= EndlBypassGeschl AND EndlBypassOffen;
		Bypassklappe.QuitFehler				:= QuitFehler;
		Bypassklappe();
		BypassOeffnenOut					:= Bypassklappe.OeffnenOut;
		BypassSchliessenOut					:= Bypassklappe.SchliessenOut;
		FehlerLaufzeitBypass				:= Bypassklappe.FehlerLaufzeitOeffnen OR Bypassklappe.FehlerLaufzeitSchliessen;
		BypassklappeIstGeschl				:= Bypassklappe.KlappeIstGeschlOut;
		BypassklappeIstOffen				:= Bypassklappe.KlappeIstOffenOut;

		Umschaltklappe1.EndlagenVhd			:= EndlagenVhdUmschaltklappe1;
		Umschaltklappe1.EndlageOffen		:= EndlUmschaltkl1Offen;
		Umschaltklappe1.EndlageGeschl		:= EndlUmschaltkl1Geschl;
		Umschaltklappe1.LaufzeitOeffnen		:= LaufzeitUmschaltklappe1;
		Umschaltklappe1.LaufzeitSchliessen	:= LaufzeitUmschaltklappe1;
		Umschaltklappe1.Stoerung			:= EndlUmschaltkl1Offen AND EndlUmschaltkl1Geschl;
		Umschaltklappe1.QuitFehler			:= QuitFehler;
		Umschaltklappe1();
		Umschaltkl1OeffnenOut				:= Umschaltklappe1.OeffnenOut;
		Umschaltkl1SchliessenOut			:= Umschaltklappe1.SchliessenOut;
		FehlerLaufzeitUmschaltkl1			:= Umschaltklappe1.FehlerLaufzeitOeffnen OR Umschaltklappe1.FehlerLaufzeitSchliessen;
		Umschaltklappe1IstGeschl			:= Umschaltklappe1.KlappeIstGeschlOut;
		Umschaltklappe1IstOffen				:= Umschaltklappe1.KlappeIstOffenOut;

		Umschaltklappe2.EndlagenVhd			:= EndlagenVhdUmschaltklappe2;
		Umschaltklappe2.EndlageOffen		:= EndlUmschaltkl2Offen;
		Umschaltklappe2.EndlageGeschl		:= EndlUmschaltkl2Geschl;
		Umschaltklappe2.LaufzeitOeffnen		:= LaufzeitUmschaltklappe2;
		Umschaltklappe2.LaufzeitSchliessen	:= LaufzeitUmschaltklappe2;
		Umschaltklappe2.Stoerung			:= EndlUmschaltkl2Offen AND EndlUmschaltkl2Geschl;
		Umschaltklappe2.QuitFehler			:= QuitFehler;
		Umschaltklappe2();
		Umschaltkl2OeffnenOut				:= Umschaltklappe2.OeffnenOut;
		Umschaltkl2SchliessenOut			:= Umschaltklappe2.SchliessenOut;
		FehlerLaufzeitUmschaltkl2			:= Umschaltklappe2.FehlerLaufzeitOeffnen OR Umschaltklappe2.FehlerLaufzeitSchliessen;
		Umschaltklappe2IstGeschl			:= Umschaltklappe2.KlappeIstGeschlOut;
		Umschaltklappe2IstOffen				:= Umschaltklappe2.KlappeIstOffenOut;

		Boxenklappe1.EndlagenVhd			:= EndlagenVhdBoxenklappe1;
		Boxenklappe1.EndlageOffen			:= EndlBoxenklappe1Offen;
		Boxenklappe1.EndlageGeschl			:= EndlBoxenklappe1Geschl;
		Boxenklappe1.LaufzeitOeffnen		:= LaufzeitBoxenklappe1;
		Boxenklappe1.LaufzeitSchliessen		:= LaufzeitBoxenklappe1;
		Boxenklappe1.Stoerung				:= EndlBoxenklappe1Offen AND EndlBoxenklappe1Geschl;
		Boxenklappe1.QuitFehler				:= QuitFehler;
		Boxenklappe1();
		Boxenklappe1IstGeschl				:= Boxenklappe1.KlappeIstGeschlOut;
		Boxenklappe1IstOffen				:= Boxenklappe1.KlappeIstOffenOut;
		IF Boxenklappe1Vorhanden THEN
			Boxenklappe1OeffnenOut				:= Boxenklappe1.OeffnenOut;
			Boxenklappe1SchliessenOut			:= Boxenklappe1.SchliessenOut;
			FehlerLaufzeitKlappeBox1			:= Boxenklappe1.FehlerLaufzeitOeffnen OR Boxenklappe1.FehlerLaufzeitSchliessen;
		ELSE
			Boxenklappe1OeffnenOut				:= FALSE;
			Boxenklappe1SchliessenOut			:= FALSE;
			FehlerLaufzeitKlappeBox1			:= FALSE;
		END_IF

		Boxenklappe2.EndlagenVhd			:= EndlagenVhdBoxenklappe2;
		Boxenklappe2.EndlageOffen			:= EndlBoxenklappe2Offen;
		Boxenklappe2.EndlageGeschl			:= EndlBoxenklappe2Geschl;
		Boxenklappe2.LaufzeitOeffnen		:= LaufzeitBoxenklappe2;
		Boxenklappe2.LaufzeitSchliessen		:= LaufzeitBoxenklappe2;
		Boxenklappe2.Stoerung				:= EndlBoxenklappe2Offen AND EndlBoxenklappe2Geschl;
		Boxenklappe2.QuitFehler				:= QuitFehler;
		Boxenklappe2();
		Boxenklappe2IstGeschl				:= Boxenklappe2.KlappeIstGeschlOut;
		Boxenklappe2IstOffen				:= Boxenklappe2.KlappeIstOffenOut;
		IF Boxenklappe2Vorhanden THEN
			Boxenklappe2OeffnenOut				:= Boxenklappe2.OeffnenOut;
			Boxenklappe2SchliessenOut			:= Boxenklappe2.SchliessenOut;
			FehlerLaufzeitKlappeBox2			:= Boxenklappe2.FehlerLaufzeitOeffnen OR Boxenklappe2.FehlerLaufzeitSchliessen;
		ELSE
			Boxenklappe2OeffnenOut				:= FALSE;
			Boxenklappe2SchliessenOut			:= FALSE;
			FehlerLaufzeitKlappeBox2			:= FALSE;
		END_IF

		Boxenklappe3.EndlagenVhd			:= EndlagenVhdBoxenklappe3;
		Boxenklappe3.EndlageOffen			:= EndlBoxenklappe3Offen;
		Boxenklappe3.EndlageGeschl			:= EndlBoxenklappe3Geschl;
		Boxenklappe3.LaufzeitOeffnen		:= LaufzeitBoxenklappe3;
		Boxenklappe3.LaufzeitSchliessen		:= LaufzeitBoxenklappe3;
		Boxenklappe3.Stoerung				:= EndlBoxenklappe3Offen AND EndlBoxenklappe3Geschl;
		Boxenklappe3.QuitFehler				:= QuitFehler;
		Boxenklappe3();
		Boxenklappe3IstGeschl				:= Boxenklappe3.KlappeIstGeschlOut;
		Boxenklappe3IstOffen				:= Boxenklappe3.KlappeIstOffenOut;
		IF Boxenklappe3Vorhanden THEN
			Boxenklappe3OeffnenOut				:= Boxenklappe3.OeffnenOut;
			Boxenklappe3SchliessenOut			:= Boxenklappe3.SchliessenOut;
			FehlerLaufzeitKlappeBox3			:= Boxenklappe3.FehlerLaufzeitOeffnen OR Boxenklappe3.FehlerLaufzeitSchliessen;
		ELSE
			Boxenklappe3OeffnenOut				:= FALSE;
			Boxenklappe3SchliessenOut			:= FALSE;
			FehlerLaufzeitKlappeBox3			:= FALSE;
		END_IF

		Boxenklappe4.EndlagenVhd			:= EndlagenVhdBoxenklappe4;
		Boxenklappe4.EndlageOffen			:= EndlBoxenklappe4Offen;
		Boxenklappe4.EndlageGeschl			:= EndlBoxenklappe4Geschl;
		Boxenklappe4.LaufzeitOeffnen		:= LaufzeitBoxenklappe4;
		Boxenklappe4.LaufzeitSchliessen		:= LaufzeitBoxenklappe4;
		Boxenklappe4.Stoerung				:= EndlBoxenklappe4Offen AND EndlBoxenklappe4Geschl;
		Boxenklappe4.QuitFehler				:= QuitFehler;
		Boxenklappe4();
		Boxenklappe4IstGeschl				:= Boxenklappe4.KlappeIstGeschlOut;
		Boxenklappe4IstOffen				:= Boxenklappe4.KlappeIstOffenOut;
		IF Boxenklappe4Vorhanden THEN
			Boxenklappe4OeffnenOut				:= Boxenklappe4.OeffnenOut;
			Boxenklappe4SchliessenOut			:= Boxenklappe4.SchliessenOut;
			FehlerLaufzeitKlappeBox4			:= Boxenklappe4.FehlerLaufzeitOeffnen OR Boxenklappe4.FehlerLaufzeitSchliessen;
		ELSE
			Boxenklappe4OeffnenOut				:= FALSE;
			Boxenklappe4SchliessenOut			:= FALSE;
			FehlerLaufzeitKlappeBox4			:= FALSE;
		END_IF

		Boxenklappe5.EndlagenVhd			:= EndlagenVhdBoxenklappe5;
		Boxenklappe5.EndlageOffen			:= EndlBoxenklappe5Offen;
		Boxenklappe5.EndlageGeschl			:= EndlBoxenklappe5Geschl;
		Boxenklappe5.LaufzeitOeffnen		:= LaufzeitBoxenklappe5;
		Boxenklappe5.LaufzeitSchliessen		:= LaufzeitBoxenklappe5;
		Boxenklappe5.Stoerung				:= EndlBoxenklappe5Offen AND EndlBoxenklappe5Geschl;
		Boxenklappe5.QuitFehler				:= QuitFehler;
		Boxenklappe5();
		Boxenklappe5IstGeschl				:= Boxenklappe5.KlappeIstGeschlOut;
		Boxenklappe5IstOffen				:= Boxenklappe5.KlappeIstOffenOut;
		IF Boxenklappe5Vorhanden THEN
			Boxenklappe5OeffnenOut				:= Boxenklappe5.OeffnenOut;
			Boxenklappe5SchliessenOut			:= Boxenklappe5.SchliessenOut;
			FehlerLaufzeitKlappeBox5			:= Boxenklappe5.FehlerLaufzeitOeffnen OR Boxenklappe5.FehlerLaufzeitSchliessen;
		ELSE
			Boxenklappe5OeffnenOut				:= FALSE;
			Boxenklappe5SchliessenOut			:= FALSE;
			FehlerLaufzeitKlappeBox5			:= FALSE;
		END_IF

		Boxenklappe6.EndlagenVhd			:= EndlagenVhdBoxenklappe6;
		Boxenklappe6.EndlageOffen			:= EndlBoxenklappe6Offen;
		Boxenklappe6.EndlageGeschl			:= EndlBoxenklappe6Geschl;
		Boxenklappe6.LaufzeitOeffnen		:= LaufzeitBoxenklappe6;
		Boxenklappe6.LaufzeitSchliessen		:= LaufzeitBoxenklappe6;
		Boxenklappe6.Stoerung				:= EndlBoxenklappe6Offen AND EndlBoxenklappe6Geschl;
		Boxenklappe6.QuitFehler				:= QuitFehler;
		Boxenklappe6();
		Boxenklappe6IstGeschl				:= Boxenklappe6.KlappeIstGeschlOut;
		Boxenklappe6IstOffen				:= Boxenklappe6.KlappeIstOffenOut;
		IF Boxenklappe6Vorhanden THEN
			Boxenklappe6OeffnenOut				:= Boxenklappe6.OeffnenOut;
			Boxenklappe6SchliessenOut			:= Boxenklappe6.SchliessenOut;
			FehlerLaufzeitKlappeBox6			:= Boxenklappe6.FehlerLaufzeitOeffnen OR Boxenklappe6.FehlerLaufzeitSchliessen;
		ELSE
			Boxenklappe6OeffnenOut				:= FALSE;
			Boxenklappe6SchliessenOut			:= FALSE;
			FehlerLaufzeitKlappeBox6			:= FALSE;
		END_IF

		//Wenn Laufzeit Klappe auf "0" (Drehzahl Ventilator wird bei Umschaltung der Klappe nicht reduziert)
		//oder Option bei Umluftklappen aktiviert -> Klappen direkt ansteuern
		IF LaufzeitBypassklappe = 0 THEN
			Bypassklappe.Oeffnen			:= BypassklappeOeffnen;
			Bypassklappe.Schliessen			:= BypassklappeSchliessen;
		END_IF
		IF (LaufzeitUmschaltklappe1 = 0) OR (NOT UmluftklVonVent1Abhaengig AND NOT UmluftklVonVent2Abhaengig) THEN
			Umschaltklappe1.Oeffnen			:= Umschaltkl1Oeffnen;
			Umschaltklappe1.Schliessen		:= Umschaltkl1Schliessen;
		END_IF
		IF (LaufzeitUmschaltklappe2 = 0) OR (NOT UmluftklVonVent1Abhaengig AND NOT UmluftklVonVent2Abhaengig) THEN
			Umschaltklappe2.Oeffnen			:= Umschaltkl2Oeffnen;
			Umschaltklappe2.Schliessen		:= Umschaltkl2Schliessen;
		END_IF
		IF LaufzeitBoxenklappe1 = 0 THEN
			Boxenklappe1.Oeffnen			:= Boxenklappe1Oeffnen AND Boxenklappe1Vorhanden;
			Boxenklappe1.Schliessen			:= Boxenklappe1Schliessen AND Boxenklappe1Vorhanden;
		END_IF
		IF LaufzeitBoxenklappe2 = 0 THEN
			Boxenklappe2.Oeffnen			:= Boxenklappe2Oeffnen AND Boxenklappe2Vorhanden;
			Boxenklappe2.Schliessen			:= Boxenklappe2Schliessen AND Boxenklappe2Vorhanden;
		END_IF
		IF LaufzeitBoxenklappe3 = 0 THEN
			Boxenklappe3.Oeffnen			:= Boxenklappe3Oeffnen AND Boxenklappe3Vorhanden;
			Boxenklappe3.Schliessen			:= Boxenklappe3Schliessen AND Boxenklappe3Vorhanden;
		END_IF
		IF LaufzeitBoxenklappe4 = 0 THEN
			Boxenklappe4.Oeffnen			:= Boxenklappe4Oeffnen AND Boxenklappe4Vorhanden;
			Boxenklappe4.Schliessen			:= Boxenklappe4Schliessen AND Boxenklappe4Vorhanden;
		END_IF
		IF LaufzeitBoxenklappe5 = 0 THEN
			Boxenklappe5.Oeffnen			:= Boxenklappe5Oeffnen AND Boxenklappe5Vorhanden;
			Boxenklappe5.Schliessen			:= Boxenklappe5Schliessen AND Boxenklappe5Vorhanden;
		END_IF
		IF LaufzeitBoxenklappe6 = 0 THEN
			Boxenklappe6.Oeffnen			:= Boxenklappe6Oeffnen AND Boxenklappe6Vorhanden;
			Boxenklappe6.Schliessen			:= Boxenklappe6Schliessen AND Boxenklappe6Vorhanden;
		END_IF

		//===============================================================================================================================================================================
		//Schrittkette
		//===============================================================================================================================================================================

		curStep	:= nextStep;

		CASE curStep OF

			//WARTEN *************************************************************************************************************************************************
			0:

				//*** state entry ***
				IF stateEntry THEN
					stateEntry 						:= FALSE;
					Bypassklappe.Oeffnen			:= FALSE;
					Bypassklappe.Schliessen			:= FALSE;
					Umschaltklappe1.Oeffnen			:= FALSE;
					Umschaltklappe1.Schliessen		:= FALSE;
					Umschaltklappe2.Oeffnen			:= FALSE;
					Umschaltklappe2.Schliessen		:= FALSE;
					Boxenklappe1.Oeffnen			:= FALSE;
					Boxenklappe1.Schliessen			:= FALSE;
					Boxenklappe2.Oeffnen			:= FALSE;
					Boxenklappe2.Schliessen			:= FALSE;
					Boxenklappe3.Oeffnen			:= FALSE;
					Boxenklappe3.Schliessen			:= FALSE;
					Boxenklappe4.Oeffnen			:= FALSE;
					Boxenklappe4.Schliessen			:= FALSE;
					Boxenklappe5.Oeffnen			:= FALSE;
					Boxenklappe5.Schliessen			:= FALSE;
					Boxenklappe6.Oeffnen			:= FALSE;
					Boxenklappe6.Schliessen			:= FALSE;
				END_IF

				//*** state during ***
				//Ventilatoren ausschalten, wenn nicht angefordert (Drehzahl zuerst auf MIN fahren)
				IF NOT AnforderungVentilator1 THEN
					fbFuVentilator1.SollDrehzahl := DrehzahlVent1Min;
					IF (fbFuVentilator1.DrehzahlFU <= DrehzahlVent1Min) AND NOT AnforderungVentilator1 THEN
						fbFuVentilator1.Freigabe := FALSE;
					END_IF
				END_IF

				IF NOT AnforderungVentilator2 THEN
					fbFuVentilator2.SollDrehzahl := DrehzahlVent2Min;
					IF (fbFuVentilator2.DrehzahlFU <= DrehzahlVent2Min) AND NOT AnforderungVentilator2 THEN
						fbFuVentilator2.Freigabe := FALSE;
					END_IF
				END_IF

			(*	IF NOT AnforderungVentilator1 THEN
					fbFuVentilator1.Freigabe		:= FALSE;
					fbFuVentilator1.SollDrehzahl	:= DrehzahlVent1Min;
				END_IF
				IF NOT AnforderungVentilator2 THEN
					fbFuVentilator2.Freigabe		:= FALSE;
					fbFuVentilator2.SollDrehzahl	:= DrehzahlVent2Min;
				END_IF*)

				//*** state exit ***
				//Ventilator 1 oder 2 angefordert und keine Umschaltung Klappen erforderlich -> VENTILATOREN EIN
				IF (AnforderungVentilator1 OR AnforderungVentilator2) AND NOT loc_UmschaltungErforderlVent1 AND NOT loc_UmschaltungErforderlVent2 THEN
					stateEntry	:= TRUE;
					lastStep	:= curStep;
					nextStep	:= 1;
					//Umschaltung Klappen erforderlich -> KLAPPEN UMSCHALTEN
				ELSIF loc_UmschaltungErforderlVent1 OR loc_UmschaltungErforderlVent2 THEN
					stateEntry	:= TRUE;
					lastStep	:= curStep;
					nextStep	:= 2;
				END_IF

			//VENTILATOREN EIN *************************************************************************************************************************************************
			1:

				//*** state entry ***
				IF stateEntry THEN
					stateEntry 						:= FALSE;
				(*	Bypassklappe.Oeffnen			:= FALSE;
					Bypassklappe.Schliessen			:= FALSE;
					Umschaltklappe1.Oeffnen			:= FALSE;
					Umschaltklappe1.Schliessen		:= FALSE;
					Umschaltklappe2.Oeffnen			:= FALSE;
					Umschaltklappe2.Schliessen		:= FALSE;
					Boxenklappe1.Oeffnen			:= FALSE;
					Boxenklappe1.Schliessen			:= FALSE;
					Boxenklappe2.Oeffnen			:= FALSE;
					Boxenklappe2.Schliessen			:= FALSE;
					Boxenklappe3.Oeffnen			:= FALSE;
					Boxenklappe3.Schliessen			:= FALSE;
					Boxenklappe4.Oeffnen			:= FALSE;
					Boxenklappe4.Schliessen			:= FALSE;
					Boxenklappe5.Oeffnen			:= FALSE;
					Boxenklappe5.Schliessen			:= FALSE;
					Boxenklappe6.Oeffnen			:= FALSE;
					Boxenklappe6.Schliessen			:= FALSE;
					TON_AnlaufverzVentilatoren(IN	:= FALSE, PT:= 0);*)
				END_IF

				//*** state during ***

				//Anlaufverzögerung Ventilatoren starten
				TON_AnlaufverzVentilatoren(IN:= AnforderungVentilator1 OR AnforderungVentilator2, PT:= AnlaufverzZweiterVent);

				//Nur 1 Ventilator angefordert
				IF (AnforderungVentilator1 AND NOT AnforderungVentilator2) OR
					(NOT AnforderungVentilator1 AND AnforderungVentilator2) THEN

					IF NOT AnforderungVentilator1 THEN
						fbFuVentilator1.SollDrehzahl := DrehzahlVent1Min;
						IF (fbFuVentilator1.DrehzahlFU <= DrehzahlVent1Min) THEN
							fbFuVentilator1.Freigabe := FALSE;
						END_IF
					ELSE
						fbFuVentilator1.Freigabe			:= AnforderungVentilator1;
						fbFuVentilator1.SollDrehzahl		:= DrehzahlVent1Betrieb;
					END_IF

					IF NOT AnforderungVentilator2 THEN
						fbFuVentilator2.SollDrehzahl := DrehzahlVent2Min;
						IF (fbFuVentilator2.DrehzahlFU <= DrehzahlVent2Min) THEN
							fbFuVentilator2.Freigabe := FALSE;
						END_IF
					ELSE
						fbFuVentilator2.Freigabe			:= AnforderungVentilator2;
						fbFuVentilator2.SollDrehzahl		:= DrehzahlVent2Betrieb;
					END_IF

					//Beide Ventilatoren angefordert
				ELSIF AnforderungVentilator1 AND AnforderungVentilator2 THEN
					IF (NOT fbFuVentilator2.Freigabe) THEN
						fbFuVentilator1.Freigabe			:= AnforderungVentilator1;
						fbFuVentilator1.SollDrehzahl		:= DrehzahlVent1Betrieb;
						IF TON_AnlaufverzVentilatoren.Q THEN
							fbFuVentilator2.Freigabe		:= AnforderungVentilator2;
							fbFuVentilator2.SollDrehzahl	:= DrehzahlVent2Betrieb;
						END_IF
					ELSIF (NOT fbFuVentilator1.Freigabe) THEN
						fbFuVentilator2.Freigabe			:= AnforderungVentilator2;
						fbFuVentilator2.SollDrehzahl		:= DrehzahlVent2Betrieb;
						IF TON_AnlaufverzVentilatoren.Q THEN
							fbFuVentilator1.Freigabe		:= AnforderungVentilator1;
							fbFuVentilator1.SollDrehzahl	:= DrehzahlVent1Betrieb;
						END_IF
					ELSE
						fbFuVentilator1.Freigabe			:= AnforderungVentilator1;
						fbFuVentilator1.SollDrehzahl		:= DrehzahlVent1Betrieb;
						IF TON_AnlaufverzVentilatoren.Q THEN
							fbFuVentilator2.Freigabe		:= AnforderungVentilator2;
							fbFuVentilator2.SollDrehzahl	:= DrehzahlVent2Betrieb;
						END_IF
					END_IF
				END_IF

				//Restzeit Anlaufverzögerung (für Visu)
				RestAnlaufverzoegerung := AnlaufverzZweiterVent - TIME_TO_UDINT(TON_AnlaufverzVentilatoren.ET);
				AnlaufverzVent1Aktiv := AnforderungVentilator1 AND (fbFuVentilator1.SollDrehzahl <> DrehzahlVent1Betrieb);
				AnlaufverzVent2Aktiv := AnforderungVentilator2 AND (fbFuVentilator2.SollDrehzahl <> DrehzahlVent2Betrieb);

				//*** state exit ***
				//Keine Anforderung von Ventilator 1 und 2 -> WARTEN
				IF (NOT AnforderungVentilator1 AND NOT AnforderungVentilator2) THEN
					stateEntry	:= TRUE;
					lastStep	:= curStep;
					nextStep	:= 0;
					//Umschaltung Klappen erforderlich -> KLAPPEN UMSCHALTEN
				ELSIF loc_UmschaltungErforderlVent1 OR loc_UmschaltungErforderlVent2 THEN
					stateEntry	:= TRUE;
					lastStep	:= curStep;
					nextStep	:= 2;
				END_IF

			//KLAPPEN UMSCHALTEN *************************************************************************************************************************************************
			2:

				//*** state entry ***

				IF stateEntry THEN
					stateEntry 						:= FALSE;
					UmschaltungAktiv				:= TRUE;
					IF loc_UmschaltungErforderlVent1 AND loc_UmschaltungErforderlVent2 THEN
						TON_AnlaufverzVentilatoren(IN:= FALSE, PT:= 0);
					END_IF
				(*	Bypassklappe.Oeffnen			:= FALSE;
					Bypassklappe.Schliessen			:= FALSE;
					Umschaltklappe1.Oeffnen			:= FALSE;
					Umschaltklappe1.Schliessen		:= FALSE;
					Umschaltklappe2.Oeffnen			:= FALSE;
					Umschaltklappe2.Schliessen		:= FALSE;
					Boxenklappe1.Oeffnen			:= FALSE;
					Boxenklappe1.Schliessen			:= FALSE;
					Boxenklappe2.Oeffnen			:= FALSE;
					Boxenklappe2.Schliessen			:= FALSE;
					Boxenklappe3.Oeffnen			:= FALSE;
					Boxenklappe3.Schliessen			:= FALSE;
					Boxenklappe4.Oeffnen			:= FALSE;
					Boxenklappe4.Schliessen			:= FALSE;
					Boxenklappe5.Oeffnen			:= FALSE;
					Boxenklappe5.Schliessen			:= FALSE;
					Boxenklappe6.Oeffnen			:= FALSE;
					Boxenklappe6.Schliessen			:= FALSE;*)
				END_IF

				//*** state during ***

				//Ventilatoren auf Min. Drehzahl fahren
				IF NOT AnforderungVentilator1 THEN
					fbFuVentilator1.SollDrehzahl := DrehzahlVent1Min;
					IF (fbFuVentilator1.DrehzahlFU <= DrehzahlVent1Min) AND NOT AnforderungVentilator1 THEN
						fbFuVentilator1.Freigabe := FALSE;
					END_IF
				END_IF

				IF NOT AnforderungVentilator2 THEN
					fbFuVentilator2.SollDrehzahl := DrehzahlVent2Min;
					IF (fbFuVentilator2.DrehzahlFU <= DrehzahlVent2Min) AND NOT AnforderungVentilator2 THEN
						fbFuVentilator2.Freigabe := FALSE;
					END_IF
				END_IF

				//Drehzahlvorgabe Ventilator 1
				IF LuftaufbereitungInBetrieb AND loc_UmschaltungErforderlVent1 THEN
					IF DrehzahlVent1Betrieb > DrzVent1UmschMitLuftaufb THEN
						fbFuVentilator1.SollDrehzahl	:= DrzVent1UmschMitLuftaufb;
					ELSE
						fbFuVentilator1.SollDrehzahl	:= DrehzahlVent1Betrieb;
					END_IF
				ELSIF loc_UmschaltungErforderlVent1 THEN
					IF DrehzahlVent1Betrieb > DrehzahlVent1Umsch THEN
						fbFuVentilator1.SollDrehzahl	:= DrehzahlVent1Umsch;
					ELSE
						fbFuVentilator1.SollDrehzahl	:= DrehzahlVent1Betrieb;
					END_IF
				END_IF

				//Drehzahlvorgabe Ventilator 2
				IF LuftaufbereitungInBetrieb AND loc_UmschaltungErforderlVent2 THEN
					IF DrehzahlVent2Betrieb > DrzVent2UmschMitLuftaufb THEN
						fbFuVentilator2.SollDrehzahl	:= DrzVent2UmschMitLuftaufb;
					ELSE
						fbFuVentilator2.SollDrehzahl	:= DrehzahlVent2Betrieb;
					END_IF
				ELSIF loc_UmschaltungErforderlVent2 THEN
					IF DrehzahlVent2Betrieb > DrehzahlVent2Umsch THEN
						fbFuVentilator2.SollDrehzahl	:= DrehzahlVent2Umsch;
					ELSE
						fbFuVentilator2.SollDrehzahl	:= DrehzahlVent2Betrieb;
					END_IF
				END_IF

				//Wenn IST-Drehzahl Ventilatoren = MIN -> Ventilatoren ausschalten
				IF (fbFuVentilator1.DrehzahlFU <= DrehzahlVent1Min) THEN
					fbFuVentilator1.Freigabe := FALSE;
				END_IF

				IF (fbFuVentilator2.DrehzahlFU <= DrehzahlVent2Min) THEN
					fbFuVentilator2.Freigabe := FALSE;
				END_IF

				//Ventilatoren Drehzahl erreicht
				IF ((fbFuVentilator1.DrehzahlFU <= fbFuVentilator1.SollDrehzahl) OR (NOT loc_UmschaltungErforderlVent1)) AND
					((fbFuVentilator2.DrehzahlFU <= fbFuVentilator2.SollDrehzahl) OR (NOT loc_UmschaltungErforderlVent2)) THEN
					Bypassklappe.Oeffnen			:= BypassklappeOeffnen;
					Bypassklappe.Schliessen			:= BypassklappeSchliessen;
					Umschaltklappe1.Oeffnen			:= Umschaltkl1Oeffnen;
					Umschaltklappe1.Schliessen		:= Umschaltkl1Schliessen;
					Umschaltklappe2.Oeffnen			:= Umschaltkl2Oeffnen;
					Umschaltklappe2.Schliessen		:= Umschaltkl2Schliessen;
					Boxenklappe1.Oeffnen			:= Boxenklappe1Oeffnen;
					Boxenklappe1.Schliessen			:= Boxenklappe1Schliessen;
					Boxenklappe2.Oeffnen			:= Boxenklappe2Oeffnen;
					Boxenklappe2.Schliessen			:= Boxenklappe2Schliessen;
					Boxenklappe3.Oeffnen			:= Boxenklappe3Oeffnen;
					Boxenklappe3.Schliessen			:= Boxenklappe3Schliessen;
					Boxenklappe4.Oeffnen			:= Boxenklappe4Oeffnen;
					Boxenklappe4.Schliessen			:= Boxenklappe4Schliessen;
					Boxenklappe5.Oeffnen			:= Boxenklappe5Oeffnen;
					Boxenklappe5.Schliessen			:= Boxenklappe5Schliessen;
					Boxenklappe6.Oeffnen			:= Boxenklappe6Oeffnen;
					Boxenklappe6.Schliessen			:= Boxenklappe6Schliessen;
				END_IF

				//*** state exit ***
				//Alle Klappen umgeschaltet -> WARTEN
				IF NOT loc_UmschaltungErforderlVent1 AND NOT loc_UmschaltungErforderlVent2 THEN
					UmschaltungAktiv := FALSE;
					stateEntry	:= TRUE;
					lastStep	:= curStep;
					nextStep	:= 0;
				END_IF

		END_CASE

	ELSE

		BypassOeffnenOut			:= FALSE;
		BypassSchliessenOut			:= FALSE;
		Umschaltkl1OeffnenOut		:= FALSE;
		Umschaltkl1SchliessenOut	:= FALSE;
		Umschaltkl2OeffnenOut		:= FALSE;
		Umschaltkl2SchliessenOut	:= FALSE;
		Boxenklappe1OeffnenOut		:= FALSE;
		Boxenklappe1SchliessenOut	:= FALSE;
		Boxenklappe2OeffnenOut		:= FALSE;
		Boxenklappe2SchliessenOut	:= FALSE;
		Boxenklappe3OeffnenOut		:= FALSE;
		Boxenklappe3SchliessenOut	:= FALSE;
		Boxenklappe4OeffnenOut		:= FALSE;
		Boxenklappe4SchliessenOut	:= FALSE;
		Boxenklappe5OeffnenOut		:= FALSE;
		Boxenklappe5SchliessenOut	:= FALSE;
		Boxenklappe6OeffnenOut		:= FALSE;
		Boxenklappe6SchliessenOut	:= FALSE;
		FreigabeVentilator1Out		:= FALSE;
		FreigabeVentilator2Out		:= FALSE;
		DrehzahlVent1Out			:= 0.0;
		DrehzahlVent2Out			:= 0.0;
		stateEntry					:= TRUE;
		curStep						:= 0;
		nextStep					:= 0;
		lastStep					:= 0;
		FehlerLaufzeitBypass		:= FALSE;
		FehlerLaufzeitKlappeBox1	:= FALSE;
		FehlerLaufzeitKlappeBox2	:= FALSE;
		FehlerLaufzeitKlappeBox3	:= FALSE;
		FehlerLaufzeitKlappeBox4	:= FALSE;
		FehlerLaufzeitKlappeBox5	:= FALSE;
		FehlerLaufzeitKlappeBox6	:= FALSE;
		FehlerLaufzeitUmschaltkl1	:= FALSE;
		FehlerLaufzeitUmschaltkl2	:= FALSE;
		FehlerFuVentilator1			:= FALSE;
		FehlerFuVentilator2			:= FALSE;
		UmschaltungAktiv			:= FALSE;

		fbFuVentilator1.Reset		:= TRUE;
		fbFuVentilator1();

		fbFuVentilator2.Reset		:= TRUE;
		fbFuVentilator2();

		Bypassklappe.QuitFehler		:= TRUE;
		Bypassklappe();

		Umschaltklappe1.QuitFehler	:= TRUE;
		Umschaltklappe1();

		Umschaltklappe2.QuitFehler	:= TRUE;
		Umschaltklappe2();

		Boxenklappe1.QuitFehler		:= TRUE;
		Boxenklappe1();

		Boxenklappe2.QuitFehler		:= TRUE;
		Boxenklappe2();

		Boxenklappe3.QuitFehler		:= TRUE;
		Boxenklappe3();

		Boxenklappe4.QuitFehler		:= TRUE;
		Boxenklappe4();

		Boxenklappe5.QuitFehler		:= TRUE;
		Boxenklappe5();

		Boxenklappe6.QuitFehler		:= TRUE;
		Boxenklappe6();

	END_IF

END_FUNCTION_BLOCK
```

#### fbBoxenKlappenanst.st
```iecst
(* Funktionsbaustein zur Ansteuerung von Klappen mit nur einem Wechsler-Relais (nicht angesteuert = Richtung A, angesteuert = Richtung B) *)
FUNCTION_BLOCK fbBoxenKlappenanst

	IF (NOT Stoerung) THEN

		//Fehlerquittierung Laufzeitüberwachung
		IF QuitFehler OR (LaufzeitOeffnen = 0) OR (NOT EndlagenVhd) THEN
			FehlerLaufzeitOeffnen		:= FALSE;
		END_IF

		IF QuitFehler OR (LaufzeitSchliessen = 0) OR (NOT EndlagenVhd) THEN
			FehlerLaufzeitSchliessen	:= FALSE;
		END_IF

		CASE step OF

			//WARTEN *****************************************************************************
			0:

				//*** state entry ***
				IF stateEntry THEN
					stateEntry		:= FALSE;
					TON_Laufzeit(IN	:= FALSE);
					TON_AnzVerz(IN	:= FALSE);
				END_IF

				//*** state during ***
				IF QuitFehler OR (LaufzeitOeffnen = 0) OR (NOT EndlagenVhd) THEN
					FehlerLaufzeitOeffnen		:= FALSE;
				END_IF

				IF QuitFehler OR (LaufzeitSchliessen = 0) OR (NOT EndlagenVhd) THEN
					FehlerLaufzeitSchliessen	:= FALSE;
				END_IF

				//*** state exit ***
				IF EndlagenVhd OR (LaufzeitOeffnen = 0) THEN
					IF Oeffnen AND NOT FehlerLaufzeitOeffnen THEN
						stateEntry	:= TRUE;
						step		:= 1;
					END_IF
				ELSE
					IF Oeffnen AND NOT KlappeIstOffenOut THEN
						stateEntry	:= TRUE;
						step		:= 1;
					END_IF
				END_IF

				IF EndlagenVhd OR (LaufzeitSchliessen = 0) THEN
					IF Schliessen AND NOT FehlerLaufzeitSchliessen THEN
						stateEntry	:= TRUE;
						step		:= 2;
					END_IF
				ELSE
					IF Schliessen AND NOT KlappeIstGeschlOut THEN
						stateEntry	:= TRUE;
						step		:= 2;
					END_IF
				END_IF

			//ÖFFNEN *****************************************************************************
			1:

				//*** state entry ***
				IF stateEntry THEN
					stateEntry		:= FALSE;
					TON_Laufzeit(IN	:= FALSE);
					TON_AnzVerz(IN	:= FALSE);
					FehlerLaufzeitOeffnen := FALSE;
					FehlerLaufzeitSchliessen := FALSE;
					SchliessenOut	:= FALSE;
					KlappeIstGeschlOut := FALSE;
					KlappeIstOffenOut := FALSE;
				END_IF

				//*** state during ***
				TON_Laufzeit(IN	:= OeffnenOut AND NOT EndlageOffen, PT:= LaufzeitOeffnen);
				TON_AnzVerz(IN := TRUE, PT := T#40ms); //V2.1.3: 40ms Anzugsverzoegerung - somit ist das andere Relaise sicher abgefallen
				OeffnenOut		:= TON_AnzVerz.Q;

				//*** state exit ***
				IF (NOT Oeffnen) OR Schliessen OR (TON_Laufzeit.Q AND (LaufzeitOeffnen <> 0)) THEN
					IF (TON_Laufzeit.Q AND (LaufzeitOeffnen <> 0) AND NOT EndlagenVhd) THEN
						KlappeIstOffenOut := TRUE;
					ELSIF (TON_Laufzeit.Q AND (LaufzeitOeffnen <> 0)) THEN
						FehlerLaufzeitOeffnen := TRUE;
					END_IF
					stateEntry	:= TRUE;
					step		:= 0;
				END_IF

				//SCHLIESSEN *****************************************************************************
			2:

				//*** state entry ***
				IF stateEntry THEN
					stateEntry		:= FALSE;
					TON_Laufzeit(IN	:= FALSE);
					TON_AnzVerz(IN	:= FALSE);
					FehlerLaufzeitOeffnen := FALSE;
					FehlerLaufzeitSchliessen := FALSE;
					OeffnenOut		:= FALSE;
					KlappeIstGeschlOut := FALSE;
					KlappeIstOffenOut := FALSE;
				END_IF

				//*** state during ***
				TON_Laufzeit(IN:= SchliessenOut AND NOT EndlageGeschl, PT:= LaufzeitSchliessen);
				TON_AnzVerz(IN := TRUE, PT := T#40ms); //V2.1.3: 40ms Anzugsverzoegerung - somit ist das andere Relaise sicher abgefallen
				SchliessenOut		:= TON_AnzVerz.Q;

				//*** state exit ***
				IF (NOT Schliessen) OR Oeffnen OR (TON_Laufzeit.Q AND (LaufzeitSchliessen <> 0)) THEN
					IF (TON_Laufzeit.Q AND (LaufzeitSchliessen <> 0) AND NOT EndlagenVhd) THEN
						KlappeIstGeschlOut := TRUE;
					ELSIF (TON_Laufzeit.Q AND (LaufzeitSchliessen <> 0)) THEN
						FehlerLaufzeitSchliessen := TRUE;
					END_IF
					stateEntry	:= TRUE;
					step		:= 0;
				END_IF

		END_CASE

	ELSE

		OeffnenOut					:= FALSE;
		SchliessenOut				:= FALSE;
		stateEntry					:= TRUE;
		FehlerLaufzeitOeffnen		:= FALSE;
		FehlerLaufzeitSchliessen	:= FALSE;
		KlappeIstGeschlOut 			:= FALSE;
		KlappeIstOffenOut 			:= FALSE;
		step						:= 0;

	END_IF

END_FUNCTION_BLOCK
```

#### fbBoxenAbluftkl.st
```iecst
(* Funktionsbaustein zur Ansteuerung Abluftklappe *)
FUNCTION_BLOCK fbBoxenAbluftkl

	IF Freigabe THEN

		CASE step OF

			//WARTEN ***************************************************************************************
			0:

				IF stateEntry THEN
					stateEntry		:= FALSE;
					TON_Laufzeit(IN	:= FALSE, PT:= 0);
				END_IF

				IF Quit OR (Laufzeit = 0) THEN
					FehlerLaufzeit	:= FALSE;
				END_IF

				IF Automatik THEN
					//Abluft Ist > Soll -> KLAPPE ÖFFNEN
					IF ((AbluftFeuchteIst + Hysterese) >= AbluftFeuchteSoll) AND NOT FehlerLaufzeit AND ((NOT EndlageOffen) OR Laufzeit = 0) THEN
						stateEntry	:= TRUE;
						step		:= 1;
					//Abluft Ist < Soll -> KLAPPE SCHLIESSEN
					ELSIF ((AbluftFeuchteIst - Hysterese) <= AbluftFeuchteSoll) AND NOT FehlerLaufzeit AND ((NOT EndlageGeschl) OR (Laufzeit = 0)) THEN
						stateEntry	:= TRUE;
						step		:= 2;
					ELSE
						step		:= step;
					END_IF
				//Handbetrieb ÖFFNEN
				ELSIF Oeffnen AND ((NOT EndlageOffen) OR (Laufzeit = 0)) THEN
					stateEntry		:= TRUE;
					step			:= 1;
				//Handbetrieb SCHLIESSEN
				ELSIF Schliessen AND ((NOT EndlageGeschl) OR (Laufzeit = 0)) THEN
					stateEntry		:= TRUE;
					step			:= 2;
				END_IF

			//ÖFFNEN *****************************************************************************************
			1:

				IF stateEntry THEN
					stateEntry		:= FALSE;
					TON_Laufzeit(IN	:= FALSE, PT:= 0);
					SchliessenOut	:= FALSE;
				END_IF

				TON_Laufzeit(IN:= OeffnenOut, PT:= Laufzeit);

				OeffnenOut		:= TRUE;

				IF (TON_Laufzeit.Q OR EndlageOffen) AND (Laufzeit <> 0) THEN
					IF TON_Laufzeit.Q THEN
						FehlerLaufzeit	:= TRUE;
					END_IF
					stateEntry		:= TRUE;
					step			:= 0;
				ELSIF ((((AbluftFeuchteIst - Hysterese) <= AbluftFeuchteSoll) AND Automatik) OR (Schliessen AND NOT Automatik)) AND (Laufzeit = 0) THEN
					stateEntry		:= TRUE;
					step			:= 0;
				ELSIF NOT Automatik AND NOT Oeffnen THEN
					stateEntry		:= TRUE;
					step			:= 0;
				END_IF

				//SCHLIESSEN *****************************************************************************************
			2:

				IF stateEntry THEN
					stateEntry		:= FALSE;
					OeffnenOut		:= FALSE;
					TON_Laufzeit(IN	:= FALSE, PT:= 0);
				END_IF

				TON_Laufzeit(IN:= SchliessenOut, PT:= Laufzeit);

				SchliessenOut	:= TRUE;

				IF (TON_Laufzeit.Q OR EndlageGeschl) AND (Laufzeit <> 0) THEN
					IF TON_Laufzeit.Q THEN
						FehlerLaufzeit	:= TRUE;
					END_IF
					stateEntry		:= TRUE;
					step			:= 0;
				ELSIF ((((AbluftFeuchteIst + Hysterese) >= AbluftFeuchteSoll) AND Automatik) OR (Oeffnen AND NOT Automatik)) AND (Laufzeit = 0) THEN
					stateEntry		:= TRUE;
					step			:= 0;
				ELSIF NOT Automatik AND NOT Schliessen THEN
					stateEntry		:= TRUE;
					step			:= 0;
				END_IF

		END_CASE

	ELSE

		OeffnenOut		:= FALSE;
		SchliessenOut	:= FALSE;
		FehlerLaufzeit	:= FALSE;
		stateEntry		:= TRUE;
		step			:= 0;

	END_IF

END_FUNCTION_BLOCK
```

#### fbBoxenAbluftvent.st
```iecst
(* Funktionsbaustein zur Ansteuerung Abluftventilator, optional mit Drehzahlvorgabe *)
FUNCTION_BLOCK fbBoxenAbluftvent

	IF Freigabe THEN

		//Zeitticks erzeugen
		fbLascoEUhr_0(Freigabe := TRUE);
		fbLascoZdxx_0(IN := fbLascoEUhr_0.Sekunde);
		sekTick	:= fbLascoZdxx_0.Q;

		//Funktionsbaustein Ansteuerung FU Abluftventilator
		fbFuAbluftventilator.AnsprechZeitFU		:= 15;
		fbFuAbluftventilator.BetrMldg			:= VentilatorInBetrieb;
		fbFuAbluftventilator.MinDrehzahl		:= DrehzahlMin;
		fbFuAbluftventilator.MaxDrehzahl		:= DrehzahlMax;
		fbFuAbluftventilator.RampeUpSek			:= RampeUp;
		fbFuAbluftventilator.RampeDownSek		:= RampeDown;
		fbFuAbluftventilator.Reset				:= QuitFehler;
		fbFuAbluftventilator.Tick				:= sekTick;
		fbFuAbluftventilator();
		FreigabeVentilatorOut					:= fbFuAbluftventilator.BetriebFU;
		DrehzahlVentilatorOut					:= fbFuAbluftventilator.DrehzahlFU;
		FehlerOut								:= fbFuAbluftventilator.StoerungFU;

		CASE step OF

			//AUS ***************************************************************************************
			0:

				IF stateEntry THEN
					stateEntry							:= FALSE;
					fbFuAbluftventilator.Freigabe		:= FALSE;
					fbFuAbluftventilator.SollDrehzahl	:= DrehzahlMin;
				END_IF

				IF QuitFehler THEN
					FehlerOut	:= FALSE;
				END_IF

				//Automatikbetrieb
				IF Automatik THEN
					stateEntry	:= TRUE;
					step		:= 1;
				//Handbetrieb EIN
				ELSIF Ein THEN
					stateEntry	:= TRUE;
					step		:= 2;
				END_IF

			//AUTOMATIKBETRIEB *****************************************************************************************
			1:

				IF stateEntry THEN
					stateEntry		:= FALSE;
				END_IF

				//Abluftfeuchte-Ist > Vorgabe -> VENTILATOR EIN
				IF ((AbluftFeuchteIst + Hysterese) >= AbluftFeuchteSoll) THEN
					fbFuAbluftventilator.Freigabe		:= TRUE;
					fbFuAbluftventilator.SollDrehzahl	:= DrehzahlSoll;
				//Abluftfeuchte-Ist < Vorgabe -> VENTILATOR AUS
				ELSIF ((AbluftFeuchteIst - Hysterese) <= AbluftFeuchteSoll) THEN
					fbFuAbluftventilator.Freigabe		:= FALSE;
					fbFuAbluftventilator.SollDrehzahl	:= DrehzahlMin;
				END_IF

				//Fehler -> AUS
				IF FehlerOut THEN
					stateEntry	:= TRUE;
					step		:= 0;
				//Handbetrieb aktiviert
				ELSIF Ein THEN
					stateEntry	:= TRUE;
					step		:= 2;
				//Keine Automatik -> AUS
				ELSIF NOT Automatik THEN
					stateEntry	:= TRUE;
					step		:= 0;
				END_IF

			//HANDBETRIEB (EIN) *****************************************************************************************
			2:

				IF stateEntry THEN
					stateEntry		:= FALSE;
				END_IF

				fbFuAbluftventilator.Freigabe		:= TRUE;
				fbFuAbluftventilator.SollDrehzahl	:= DrehzahlSoll;

				//Fehler -> AUS
				IF FehlerOut THEN
					stateEntry	:= TRUE;
					step		:= 0;
				//Automatik aktiviert
				ELSIF Automatik THEN
					stateEntry	:= TRUE;
					step		:= 1;
				//Kein Handbetrieb -> AUS
				ELSIF NOT Ein THEN
					stateEntry	:= TRUE;
					step		:= 0;
				END_IF

		END_CASE

	ELSE

		FreigabeVentilatorOut		:= FALSE;
		DrehzahlVentilatorOut		:= 0.0;
		FehlerOut					:= FALSE;
		stateEntry					:= TRUE;
		step						:= 0;

	END_IF

END_FUNCTION_BLOCK
```

#### fbBoxenUmschaltung.st
```iecst
(* Funktionsbaustein für Umschaltung Frischluft/Umluft *)
FUNCTION_BLOCK fbBoxenUmschaltung

	IF Freigabe THEN

		CASE step OF

			//WARTEN ****************************************************************************************************************************
			0:

				//*** state entry ***
				IF stateEntry THEN
					stateEntry	:= FALSE;
				END_IF

				//*** state during ***
				//Fehler Frischluft- und Dachluftsensor -> UMLUFT
				IF NOT StatusSensorDachluftOk AND NOT StatusSensorFrischluftOk THEN
					UmluftbetriebOut		:= TRUE;
					FrischluftbetriebOut	:= FALSE;
				//Frischluft- und Dachluftsensor nicht vorhanden -> UMLUFT
				ELSIF NOT SensorDachluftVhd AND NOT SensorFrischluftVhd THEN
					UmluftbetriebOut		:= TRUE;
					FrischluftbetriebOut	:= FALSE;
				//Fehler Frischluftsensor und Dachluftsensor nicht vorhanden -> UMLUFT
				ELSIF SensorFrischluftVhd AND NOT StatusSensorFrischluftOk AND NOT SensorDachluftVhd THEN
					UmluftbetriebOut		:= TRUE;
					FrischluftbetriebOut	:= FALSE;
				//Fehler Dachluftsensor und Frischluftsensor nicht vorhanden -> UMLUFT
				ELSIF SensorDachluftVhd AND NOT StatusSensorDachluftOk AND NOT SensorFrischluftVhd THEN
					UmluftbetriebOut		:= TRUE;
					FrischluftbetriebOut	:= FALSE;
				//Frischluft- und Dachluftsensor vorhanden, beide Sensoren Fehler -> UMLUFT
				ELSIF SensorDachluftVhd AND SensorFrischluftVhd AND NOT StatusSensorDachluftOk AND NOT StatusSensorFrischluftOk THEN
					UmluftbetriebOut		:= TRUE;
					FrischluftbetriebOut	:= FALSE;
				END_IF

				//*** state exit ***
				//Abluft- und Dachluftsensor vorhanden -> Umschaltung nach Differenz Abluft/Dachluft
				IF SensorAbluftVhd AND SensorDachluftVhd AND StatusSensorAbluftOk AND StatusSensorDachluftOk THEN
					stateEntry	:= TRUE;
					step		:= 1;
				//Abluft- und Frischluftsensor vorhanden -> Umschaltung nach Differenz Abluft/Frischluft
				ELSIF SensorAbluftVhd AND SensorFrischluftVhd AND StatusSensorAbluftOk AND StatusSensorFrischluftOk THEN
					stateEntry	:= TRUE;
					step		:= 2;
				//Dachluftsensor vorhanden -> Umschaltung nach fixem Temperaturwert Dach
				ELSIF (SensorDachluftVhd AND StatusSensorDachluftOk) THEN
					stateEntry	:= TRUE;
					step		:= 3;
				//Nur Frischluftsensor vorhanden -> Umschaltung nach fixem Temperaturwert Frischluft
				ELSIF (SensorFrischluftVhd AND StatusSensorFrischluftOk) THEN
					stateEntry	:= TRUE;
					step		:= 4;
				END_IF

			//SENSOR ABLUFT UND DACHLUFT VORHANDEN ****************************************************************************************************************************
			1:
				//*** state entry ***
				IF stateEntry THEN
					stateEntry	:= FALSE;
				END_IF

				//*** state during ***

				//Bei Neustart (Kein Frischluftbetrieb, kein Umluftbetrieb) ohne Verzögerung umschalten
				IF NOT FrischluftbetriebOut AND NOT UmluftbetriebOut THEN
					IF (DachluftTemp <= AbluftTemp) THEN
						UmluftbetriebOut	:= TRUE;
					ELSIF ((DachluftTemp + DifferenzTempUmschaltung) >= AbluftTemp) THEN
						FrischluftbetriebOut	:= TRUE;
					ELSE
						UmluftbetriebOut	:= TRUE;
					END_IF
				END_IF

				//Umschaltverzögerung Frischluft/Umluft
				TON_Umluft(IN:= FrischluftbetriebOut AND (DachluftTemp <= AbluftTemp), PT:= Umschaltverz);
				TON_Frischluft(IN:= UmluftbetriebOut AND (DachluftTemp > (AbluftTemp + DifferenzTempUmschaltung)), PT:= Umschaltverz);

				IF EDGEPOS(TON_Umluft.Q) THEN
					UmluftbetriebOut		:= TRUE;
					FrischluftbetriebOut	:= FALSE;
				ELSIF EDGEPOS(TON_Frischluft.Q) THEN
					UmluftbetriebOut		:= FALSE;
					FrischluftbetriebOut	:= TRUE;
				END_IF

				//*** state exit ***
				IF (NOT SensorAbluftVhd) OR (NOT SensorDachluftVhd) OR (NOT StatusSensorDachluftOk) OR (NOT StatusSensorAbluftOk) THEN
					stateEntry	:= TRUE;
					step		:= 0;
				END_IF

			//SENSOR ABLUFT UND FRISCHLUFT VORHANDEN ****************************************************************************************************************************
			2:
				//*** state entry ***
				IF stateEntry THEN
					stateEntry	:= FALSE;
				END_IF

				//*** state during ***

				//Bei Neustart (Kein Frischluftbetrieb, kein Umluftbetrieb) ohne Verzögerung umschalten
				IF NOT FrischluftbetriebOut AND NOT UmluftbetriebOut THEN
					IF (FrischluftTemp <= AbluftTemp) THEN
						UmluftbetriebOut	:= TRUE;
					ELSIF ((FrischluftTemp + DifferenzTempUmschaltung) >= AbluftTemp) THEN
						FrischluftbetriebOut	:= TRUE;
					ELSE
						UmluftbetriebOut	:= TRUE;
					END_IF
				END_IF

				//Umschaltverzögerung Frischluft/Umluft
				TON_Umluft(IN:= FrischluftbetriebOut AND (FrischluftTemp <= AbluftTemp), PT:= Umschaltverz);
				TON_Frischluft(IN:= UmluftbetriebOut AND (FrischluftTemp > (AbluftTemp + DifferenzTempUmschaltung)), PT:= Umschaltverz);

				IF EDGEPOS(TON_Umluft.Q) THEN
					UmluftbetriebOut		:= TRUE;
					FrischluftbetriebOut	:= FALSE;
				ELSIF EDGEPOS(TON_Frischluft.Q) THEN
					UmluftbetriebOut		:= FALSE;
					FrischluftbetriebOut	:= TRUE;
				END_IF

				//*** state exit ***
				IF (NOT SensorAbluftVhd) OR (NOT SensorFrischluftVhd) OR (NOT StatusSensorFrischluftOk) OR (NOT StatusSensorAbluftOk) THEN
					stateEntry	:= TRUE;
					step		:= 0;
				END_IF

			//SENSOR DACHLUFT VORHANDEN ****************************************************************************************************************************
			3:
				//*** state entry ***
				IF stateEntry THEN
					stateEntry	:= FALSE;
				END_IF

				//*** state during ***

				//Bei Neustart (Kein Frischluftbetrieb, kein Umluftbetrieb) ohne Verzögerung umschalten
				IF NOT FrischluftbetriebOut AND NOT UmluftbetriebOut THEN
					IF (DachluftTemp <= FrischlDachlTempUmschaltung) THEN
						UmluftbetriebOut	:= TRUE;
					ELSIF (DachluftTemp >= FrischlDachlTempUmschaltung) THEN
						FrischluftbetriebOut	:= TRUE;
					ELSE
						UmluftbetriebOut	:= TRUE;
					END_IF
				END_IF

				//Umschaltverzögerung Frischluft/Umluft
				TON_Umluft(IN:= FrischluftbetriebOut AND (DachluftTemp <= (FrischlDachlTempUmschaltung - Hysterese)), PT:= Umschaltverz);
				TON_Frischluft(IN:= UmluftbetriebOut AND (DachluftTemp > FrischlDachlTempUmschaltung), PT:= Umschaltverz);

				IF EDGEPOS(TON_Umluft.Q) THEN
					UmluftbetriebOut		:= TRUE;
					FrischluftbetriebOut	:= FALSE;
				ELSIF EDGEPOS(TON_Frischluft.Q) THEN
					UmluftbetriebOut		:= FALSE;
					FrischluftbetriebOut	:= TRUE;
				END_IF

				//*** state exit ***
				IF (NOT SensorDachluftVhd) OR (NOT StatusSensorDachluftOk) THEN
					stateEntry	:= TRUE;
					step		:= 0;
				END_IF

			//NUR SENSOR FRISCHLUFT VORHANDEN ****************************************************************************************************************************
			4:
				//*** state entry ***
				IF stateEntry THEN
					stateEntry	:= FALSE;
				END_IF

				//*** state during ***

				//Bei Neustart (Kein Frischluftbetrieb, kein Umluftbetrieb) ohne Verzögerung umschalten
				IF NOT FrischluftbetriebOut AND NOT UmluftbetriebOut THEN
					IF (FrischluftTemp <= FrischlDachlTempUmschaltung) THEN
						UmluftbetriebOut	:= TRUE;
					ELSIF (FrischluftTemp >= FrischlDachlTempUmschaltung) THEN
						FrischluftbetriebOut	:= TRUE;
					END_IF
				END_IF

				//Umschaltverzögerung Frischluft/Umluft
				TON_Umluft(IN:= FrischluftbetriebOut AND (FrischluftTemp <= (FrischlDachlTempUmschaltung - Hysterese)), PT:= Umschaltverz);
				TON_Frischluft(IN:= UmluftbetriebOut AND (FrischluftTemp > FrischlDachlTempUmschaltung), PT:= Umschaltverz);

				IF EDGEPOS(TON_Umluft.Q) THEN
					UmluftbetriebOut		:= TRUE;
					FrischluftbetriebOut	:= FALSE;
				ELSIF EDGEPOS(TON_Frischluft.Q) THEN
					UmluftbetriebOut		:= FALSE;
					FrischluftbetriebOut	:= TRUE;
				END_IF

				//*** state exit ***
				IF (NOT SensorFrischluftVhd) OR (NOT StatusSensorFrischluftOk) THEN
					stateEntry	:= TRUE;
					step		:= 0;
				END_IF

		END_CASE

	ELSE

		stateEntry				:= TRUE;
		step					:= 0;
		FrischluftbetriebOut	:= TRUE;
		UmluftbetriebOut		:= FALSE;

	END_IF

END_FUNCTION_BLOCK
```

#### fbBoxenWLO.st
```iecst
(* Funktionsbaustein zur Ansteuerung Warmluftofen inkl. Solltemperatur-Vorgabe *)
FUNCTION_BLOCK fbBoxenWLO

	//Auskühlzeit Warmluftofen, wenn Option Betriebsmeldung nicht vorhanden
	TOF_Auskuehlzeit(IN:= FreigabeWarmluftofenOut, PT:= Auskuehlzeit);

	//Restlaufzeit Auskühlung berechnen (für Visu)
	RestAuskuehlzeit	:= Auskuehlzeit - TIME_TO_UDINT(TOF_Auskuehlzeit.ET);

	//Ausgang für Warmluftofen aktiv
	WarmluftofenAktiv	:= (TOF_Auskuehlzeit.Q AND NOT OptionBetriebsmldgVhd) OR (BetriebsmeldungWarmluftofen  AND OptionBetriebsmldgVhd) OR FreigabeWarmluftofenOut;

	//Fehlerquittierung
	IF QuitFehler THEN
		FehlerSensorAussenluftOut	:= FALSE;
		FehlerBetriebsmeldungOut	:= FALSE;
	END_IF

	IF Freigabe THEN

		CASE step OF

			//AUS *********************************************************************************************************************************************************
			0:

				IF stateEntry THEN
					stateEntry					:= FALSE;
					FreigabeWarmluftofenOut		:= FALSE;
					WarmlufttempSollOut			:= 0.0;
					TON_VerzBetriebsmeldung(IN	:= FALSE, PT:= 0);
				END_IF

				//Autmatikbetrieb aktiviert
				IF Automatikbetrieb AND NOT FehlerSensorAussenluftOut AND NOT FehlerBetriebsmeldungOut AND NOT FehlerSensorAussenluft THEN
					stateEntry	:= TRUE;
					step		:= 1;
				ELSIF Dauerbetrieb AND NOT FehlerSensorAussenluftOut AND NOT FehlerBetriebsmeldungOut THEN
					stateEntry	:= TRUE;
					step		:= 2;
				END_IF

				//AUTOMATIKBETRIEB *********************************************************************************************************************************************************
			1:

				IF stateEntry THEN
					stateEntry					:= FALSE;
					TON_VerzBetriebsmeldung(IN	:= FALSE, PT:= 0);
				END_IF

				//Bei Neustart (Wetter nicht gut oder schlecht) ohne Verzögerung umschalten
				IF NOT loc_WetterIstSchlecht AND NOT loc_WetterIstGut THEN
					IF (FrischluftSattDefizitIst < FrischluftSattDefizitSoll) THEN
						loc_WetterIstSchlecht	:= TRUE;
					ELSIF (FrischluftSattDefizitIst >= FrischluftSattDefizitSoll) THEN
						loc_WetterIstGut	:= TRUE;
					END_IF
				END_IF

				//Umschaltverzögerung gutes Wetter/ schlechtes Wetter
				TON_WetterIstGut(IN:= loc_WetterIstSchlecht AND (FrischluftSattDefizitIst >= (FrischluftSattDefizitSoll + Hysterese)), PT:= UmschaltverzWitterung);
				TON_WetterIstSchlecht(IN:= loc_WetterIstGut AND (FrischluftSattDefizitIst < (FrischluftSattDefizitSoll - Hysterese)), PT:= UmschaltverzWitterung);

				IF EDGEPOS(TON_WetterIstGut.Q) THEN
					loc_WetterIstGut		:= TRUE;
					loc_WetterIstSchlecht	:= FALSE;
				ELSIF EDGEPOS(TON_WetterIstSchlecht.Q) THEN
					loc_WetterIstGut		:= FALSE;
					loc_WetterIstSchlecht	:= TRUE;
				END_IF

				//Freigabe Warmluftofen
				FreigabeWarmluftofenOut	:= loc_WetterIstSchlecht OR WetterIstSchlecht;
				WarmlufttempSollOut		:= WarmlufttemperaturVorgabe;

				//Verzögerung Überwachung Betriebsmeldung (Zündzeit)
				TON_VerzBetriebsmeldung(IN:= FreigabeWarmluftofenOut AND OptionBetriebsmldgVhd AND NOT BetriebsmeldungWarmluftofen, PT:= VerzBetriebsmeldung);

				//Fehler keine Betriebsmeldung
				IF TON_VerzBetriebsmeldung.Q THEN
					FehlerBetriebsmeldungOut := TRUE;
					stateEntry	:= TRUE;
					step		:= 0;
				//Fehler Sensor Frischluft
				ELSIF FehlerSensorAussenluft THEN
					FehlerSensorAussenluftOut := TRUE;
					stateEntry	:= TRUE;
					step		:= 0;
					//Dauerbetrieb Aktiv
				ELSIF Dauerbetrieb THEN
					stateEntry	:= TRUE;
					step		:= 2;
					//Kein Automatikbetrieb
				ELSIF NOT Automatikbetrieb THEN
					stateEntry	:= TRUE;
					step		:= 0;
				END_IF

				//DAUERBETRIEB *********************************************************************************************************************************************************
			2:

				IF stateEntry THEN
					stateEntry					:= FALSE;
					TON_VerzBetriebsmeldung(IN	:= FALSE, PT:= 0);
				END_IF

				//Freigabe Warmluftofen
				FreigabeWarmluftofenOut	:= TRUE;
				WarmlufttempSollOut		:= WarmlufttemperaturVorgabe;

				//Verzögerung Überwachung Betriebsmeldung (Zündzeit)
				TON_VerzBetriebsmeldung(IN:= FreigabeWarmluftofenOut AND OptionBetriebsmldgVhd AND NOT BetriebsmeldungWarmluftofen, PT:= VerzBetriebsmeldung);

				//Fehler
				IF TON_VerzBetriebsmeldung.Q THEN
					FehlerBetriebsmeldungOut := TRUE;
					stateEntry	:= TRUE;
					step		:= 0;
					//Automatikbetrieb Aktiv
				ELSIF Automatikbetrieb THEN
					stateEntry	:= TRUE;
					step		:= 1;
					//Kein Dauerbetrieb
				ELSIF NOT Dauerbetrieb THEN
					stateEntry	:= TRUE;
					step		:= 0;
				END_IF

		END_CASE

	ELSE

		FreigabeWarmluftofenOut		:= FALSE;
		WarmlufttemperaturVorgabe	:= 0.0;
		step						:= 0;
		stateEntry					:= TRUE;
		FehlerSensorAussenluftOut	:= FALSE;
		FehlerBetriebsmeldungOut	:= FALSE;

	END_IF

END_FUNCTION_BLOCK
```

#### fbBoxenHeizreg.st
```iecst
(* Funktionsbaustein zur Ansteuerung eines Heizregisters inkl. Drehzahlvorgabe Heizungspumpe *)
FUNCTION_BLOCK fbBoxenHeizreg

	IF Freigabe THEN

		//Fehlerquittierung
		IF QuitFehler THEN
			FehlerOut	:= FALSE;
		END_IF

		CASE step OF

			//AUS *********************************************************************************************************************************************************
			0:

				IF stateEntry THEN
					stateEntry					:= FALSE;
					FreigabeHeizregisterOut		:= FALSE;
					DrehzahlHeizregisterOut		:= 0.0;
				END_IF

				//Autmatikbetrieb aktiviert
				IF Automatikbetrieb AND NOT FehlerOut AND NOT FehlerSensorAussenluft THEN
					stateEntry	:= TRUE;
					step		:= 1;
				ELSIF Dauerbetrieb AND NOT FehlerOut THEN
					stateEntry	:= TRUE;
					step		:= 2;
				END_IF

			//AUTOMATIKBETRIEB *********************************************************************************************************************************************************
			1:

				IF stateEntry THEN
					stateEntry	:= FALSE;
				END_IF

				//Bei Neustart (Wetter nicht gut oder schlecht) ohne Verzögerung umschalten
				IF NOT loc_WetterIstSchlecht AND NOT loc_WetterIstGut THEN
					IF (FrischluftSattDefizitIst < FrischluftSattDefizitSoll) THEN
						loc_WetterIstSchlecht	:= TRUE;
					ELSIF (FrischluftSattDefizitIst >= FrischluftSattDefizitSoll) THEN
						loc_WetterIstGut	:= TRUE;
					END_IF
				END_IF

				//Umschaltverzögerung gutes Wetter/ schlechtes Wetter
				TON_WetterIstGut(IN:= loc_WetterIstSchlecht AND (FrischluftSattDefizitIst >= (FrischluftSattDefizitSoll + Hysterese)), PT:= UmschaltverzWitterung);
				TON_WetterIstSchlecht(IN:= loc_WetterIstGut AND (FrischluftSattDefizitIst < (FrischluftSattDefizitSoll - Hysterese)), PT:= UmschaltverzWitterung);

				IF EDGEPOS(TON_WetterIstGut.Q) THEN
					loc_WetterIstGut		:= TRUE;
					loc_WetterIstSchlecht	:= FALSE;
				ELSIF EDGEPOS(TON_WetterIstSchlecht.Q) THEN
					loc_WetterIstGut		:= FALSE;
					loc_WetterIstSchlecht	:= TRUE;
				END_IF

				//Freigabe Heizregister
				FreigabeHeizregisterOut		:= loc_WetterIstSchlecht OR WetterIstSchlecht;
				DrehzahlHeizregisterOut		:= DrehzahlHeizregisterSoll;

				//Fehler
				IF FehlerSensorAussenluft THEN
					FehlerOut	:= TRUE;
					stateEntry	:= TRUE;
					step		:= 0;
				//Dauerbetrieb Aktiv
				ELSIF Dauerbetrieb THEN
					stateEntry	:= TRUE;
					step		:= 2;
					//Kein Automatikbetrieb
				ELSIF NOT Automatikbetrieb THEN
					stateEntry	:= TRUE;
					step		:= 0;
				END_IF

				//DAUERBETRIEB *********************************************************************************************************************************************************
			2:

				IF stateEntry THEN
					stateEntry		:= FALSE;
				END_IF

				//Freigabe Heizregister
				FreigabeHeizregisterOut		:= TRUE;
				DrehzahlHeizregisterOut		:= DrehzahlHeizregisterSoll;

				//Automatikbetrieb Aktiv
				IF Automatikbetrieb THEN
					stateEntry	:= TRUE;
					step		:= 1;
				//Kein Dauerbetrieb
				ELSIF NOT Dauerbetrieb THEN
					stateEntry	:= TRUE;
					step		:= 0;
				END_IF

		END_CASE

	ELSE

		FreigabeHeizregisterOut		:= FALSE;
		DrehzahlHeizregisterOut		:= 0.0;
		step						:= 0;
		stateEntry					:= TRUE;
		FehlerOut					:= FALSE;

	END_IF

END_FUNCTION_BLOCK
```

#### fbBoxenNotstrom.st
```iecst
(* Funktionsbaustein zur Ansteuerung eines Notstromaggregates inkl. Vorlaufzeit und Abfrage Betriebsmeldung *)
FUNCTION_BLOCK fbBoxenNotstrom

	IF Freigabe THEN

		//Verzögerung Abfrage Betriebsmeldung Notstromaggregat, Fehler bilden wenn Zeit abgelaufen
		TON_VerzBetriebsmeldung(IN:= NotstromaggregatAngefordert AND (VerzBetriebsmeldung <> 0) AND NOT BetriebsmldgNotstromaggregat AND NOT QuitFehler, PT:= VerzBetriebsmeldung);
		FehlerOut	:= TON_VerzBetriebsmeldung.Q;

		//Nachlaufzeit Notstromaggregat
		TOF_Nachlaufzeit(IN:= FreigabeNotstromaggregatOut, PT:= Nachlaufzeit);

		//Freigabe Notstromaggregat, wenn Angefordert und Laufzeitüberwachung Betriebsmeldung nicht ausgelöst
		FreigabeNotstromaggregatOut	:= NotstromaggregatAngefordert AND NOT FehlerOut;

		//Ausgabe Notstrom bereit, wenn Vorlaufzeit abgelaufen
		TON_Vorlaufzeit(IN:= FreigabeNotstromaggregatOut AND (BetriebsmldgNotstromaggregat OR (VerzBetriebsmeldung = 0)), PT:= Vorlaufzeit);
		NotstromBereitOut	:= TON_Vorlaufzeit.Q AND (BetriebsmldgNotstromaggregat OR (VerzBetriebsmeldung = 0));

		//Rest Vorlaufzeit & Nachlaufzeit Notstromaggregat (für Visu)
		RestVorlaufzeit := Vorlaufzeit - TIME_TO_UDINT(TON_Vorlaufzeit.ET);
		RestNachlaufzeit := Nachlaufzeit - TIME_TO_UDINT(TOF_Nachlaufzeit.ET);

	ELSE

		FreigabeNotstromaggregatOut	:= FALSE;
		FehlerOut					:= FALSE;
		NotstromBereitOut			:= FALSE;
		TON_VerzBetriebsmeldung(IN	:= FALSE, PT:= 0);
		TON_Vorlaufzeit(IN			:= FALSE, PT:= 0);

	END_IF

END_FUNCTION_BLOCK
```

#### fbBoxenSHO.st
```iecst
(* Funktionsbaustein Ansteuerung Scheitholzofen (Auskühlzeit) *)
FUNCTION_BLOCK fbBoxenSHO

	IF Freigabe THEN

		TOF_Auskuehlzeit(IN:= Betriebsmeldung, PT:= Auskuehlzeit);

		//Restlaufzeit Auskühlung berechnen (für Visu)
		RestAuskuehlzeit	:= Auskuehlzeit - TIME_TO_UDINT(TOF_Auskuehlzeit.ET);

		ScheitholzofenAktiv	:= TOF_Auskuehlzeit.Q;

	ELSE

		TOF_Auskuehlzeit(IN:= FALSE, PT:= 0);
		ScheitholzofenAktiv	:= FALSE;

	END_IF

END_FUNCTION_BLOCK
```

#### fbBoxenLuftmengen.st
```iecst
(* Funktionsblock zur Ermittlung der erforderlichen Luftmengen für Ventilator 1&2 aus Boxenfläche *)
FUNCTION_BLOCK fbBoxenLuftmengen

	//Min/Max Luftmenge bei Betrieb mit Entfeuchter ermitteln
	loc_MinLuftmengeMitEntfeuchter	:= LuftgeschwEntfeuchterMin * RegisterflaecheEntfeuchter * 3600;
	loc_MaxLuftmengeMitEntfeuchter	:= LuftgeschwEntfeuchterMax * RegisterflaecheEntfeuchter * 3600;

	//Soll-Luftmenge Ventilator 1 *********************************************************************************************************************************************
	loc_LuftmengeSollVent1	:= 0;

	IF FrischluftbetriebAktiv THEN
		IF Box1.BoxIstAktiv AND Box1.Ventilator1 THEN
			loc_LuftmengeSollVent1	:= Box1.GrundflaecheBox * LuftmengeSollProM2FrischlVent1;
		END_IF
		IF Box2.BoxIstAktiv AND Box2.Ventilator1 THEN
			loc_LuftmengeSollVent1	:= loc_LuftmengeSollVent1 + (Box2.GrundflaecheBox * LuftmengeSollProM2FrischlVent1);
		END_IF
		IF Box3.BoxIstAktiv AND Box3.Ventilator1 THEN
			loc_LuftmengeSollVent1	:= loc_LuftmengeSollVent1 + (Box3.GrundflaecheBox * LuftmengeSollProM2FrischlVent1);
		END_IF
		IF Box4.BoxIstAktiv AND Box4.Ventilator1 THEN
			loc_LuftmengeSollVent1	:= loc_LuftmengeSollVent1 + (Box4.GrundflaecheBox * LuftmengeSollProM2FrischlVent1);
		END_IF
		IF Box5.BoxIstAktiv AND Box5.Ventilator1 THEN
			loc_LuftmengeSollVent1	:= loc_LuftmengeSollVent1 + (Box5.GrundflaecheBox * LuftmengeSollProM2FrischlVent1);
		END_IF
		IF Box6.BoxIstAktiv AND Box6.Ventilator1 THEN
			loc_LuftmengeSollVent1	:= loc_LuftmengeSollVent1 + (Box6.GrundflaecheBox * LuftmengeSollProM2FrischlVent1);
		END_IF
	ELSIF UmluftbetriebAktiv THEN
		IF Box1.BoxIstAktiv AND Box1.Ventilator1 THEN
			loc_LuftmengeSollVent1	:= Box1.GrundflaecheBox * LuftmengeSollProM2UmluftVent1;
		END_IF
		IF Box2.BoxIstAktiv AND Box2.Ventilator1 THEN
			loc_LuftmengeSollVent1	:= loc_LuftmengeSollVent1 + (Box2.GrundflaecheBox * LuftmengeSollProM2UmluftVent1);
		END_IF
		IF Box3.BoxIstAktiv AND Box3.Ventilator1 THEN
			loc_LuftmengeSollVent1	:= loc_LuftmengeSollVent1 + (Box3.GrundflaecheBox * LuftmengeSollProM2UmluftVent1);
		END_IF
		IF Box4.BoxIstAktiv AND Box4.Ventilator1 THEN
			loc_LuftmengeSollVent1	:= loc_LuftmengeSollVent1 + (Box4.GrundflaecheBox * LuftmengeSollProM2UmluftVent1);
		END_IF
		IF Box5.BoxIstAktiv AND Box5.Ventilator1 THEN
			loc_LuftmengeSollVent1	:= loc_LuftmengeSollVent1 + (Box5.GrundflaecheBox * LuftmengeSollProM2UmluftVent1);
		END_IF
		IF Box6.BoxIstAktiv AND Box6.Ventilator1 THEN
			loc_LuftmengeSollVent1	:= loc_LuftmengeSollVent1 + (Box6.GrundflaecheBox * LuftmengeSollProM2UmluftVent1);
		END_IF
	END_IF

	//Wenn Entfeuchter in Betrieb -> Luftmenge auf Min/Max von Entfeuchter begrenzen
	IF EntfeuchterInBetrieb THEN
		IF loc_LuftmengeSollVent1 < loc_MinLuftmengeMitEntfeuchter THEN
			LuftmengeSollVent1Out	:= loc_MinLuftmengeMitEntfeuchter;
		ELSIF loc_LuftmengeSollVent1 > loc_MaxLuftmengeMitEntfeuchter THEN
			LuftmengeSollVent1Out	:= loc_MaxLuftmengeMitEntfeuchter;
		ELSE
			LuftmengeSollVent1Out	:= loc_LuftmengeSollVent1;
		END_IF
	ELSE
		LuftmengeSollVent1Out	:= loc_LuftmengeSollVent1;
	END_IF

	//Soll-Luftmenge Ventilator 2 *********************************************************************************************************************************************
	loc_LuftmengeSollVent2	:= 0;

	IF FrischluftbetriebAktiv THEN
		IF Box1.BoxIstAktiv AND Box1.Ventilator2 THEN
			loc_LuftmengeSollVent2	:= Box1.GrundflaecheBox * LuftmengeSollProM2FrischlVent2;
		END_IF
		IF Box2.BoxIstAktiv AND Box2.Ventilator2 THEN
			loc_LuftmengeSollVent2	:= loc_LuftmengeSollVent2 + (Box2.GrundflaecheBox * LuftmengeSollProM2FrischlVent2);
		END_IF
		IF Box3.BoxIstAktiv AND Box3.Ventilator2 THEN
			loc_LuftmengeSollVent2	:= loc_LuftmengeSollVent2 + (Box3.GrundflaecheBox * LuftmengeSollProM2FrischlVent2);
		END_IF
		IF Box4.BoxIstAktiv AND Box4.Ventilator2 THEN
			loc_LuftmengeSollVent2	:= loc_LuftmengeSollVent2 + (Box4.GrundflaecheBox * LuftmengeSollProM2FrischlVent2);
		END_IF
		IF Box5.BoxIstAktiv AND Box5.Ventilator2 THEN
			loc_LuftmengeSollVent2	:= loc_LuftmengeSollVent2 + (Box5.GrundflaecheBox * LuftmengeSollProM2FrischlVent2);
		END_IF
		IF Box6.BoxIstAktiv AND Box6.Ventilator2 THEN
			loc_LuftmengeSollVent2	:= loc_LuftmengeSollVent2 + (Box6.GrundflaecheBox * LuftmengeSollProM2FrischlVent2);
		END_IF
	ELSIF UmluftbetriebAktiv THEN
		IF Box1.BoxIstAktiv AND Box1.Ventilator2 THEN
			loc_LuftmengeSollVent2	:= Box1.GrundflaecheBox * LuftmengeSollProM2UmluftVent2;
		END_IF
		IF Box2.BoxIstAktiv AND Box2.Ventilator2 THEN
			loc_LuftmengeSollVent2	:= loc_LuftmengeSollVent2 + (Box2.GrundflaecheBox * LuftmengeSollProM2UmluftVent2);
		END_IF
		IF Box3.BoxIstAktiv AND Box3.Ventilator2 THEN
			loc_LuftmengeSollVent2	:= loc_LuftmengeSollVent2 + (Box3.GrundflaecheBox * LuftmengeSollProM2UmluftVent2);
		END_IF
		IF Box4.BoxIstAktiv AND Box4.Ventilator2 THEN
			loc_LuftmengeSollVent2	:= loc_LuftmengeSollVent2 + (Box4.GrundflaecheBox * LuftmengeSollProM2UmluftVent2);
		END_IF
		IF Box5.BoxIstAktiv AND Box5.Ventilator2 THEN
			loc_LuftmengeSollVent2	:= loc_LuftmengeSollVent2 + (Box5.GrundflaecheBox * LuftmengeSollProM2UmluftVent2);
		END_IF
		IF Box6.BoxIstAktiv AND Box6.Ventilator2 THEN
			loc_LuftmengeSollVent2	:= loc_LuftmengeSollVent2 + (Box6.GrundflaecheBox * LuftmengeSollProM2UmluftVent2);
		END_IF
	END_IF

	//Wenn Entfeuchter in Betrieb -> Luftmenge auf Min/Max von Entfeuchter begrenzen
	IF EntfeuchterInBetrieb THEN
		IF loc_LuftmengeSollVent2 < loc_MinLuftmengeMitEntfeuchter THEN
			LuftmengeSollVent2Out	:= loc_MinLuftmengeMitEntfeuchter;
		ELSIF loc_LuftmengeSollVent2 > loc_MaxLuftmengeMitEntfeuchter THEN
			LuftmengeSollVent2Out	:= loc_MaxLuftmengeMitEntfeuchter;
		ELSE
			LuftmengeSollVent2Out	:= loc_LuftmengeSollVent2;
		END_IF
	ELSE
		LuftmengeSollVent2Out	:= loc_LuftmengeSollVent2;
	END_IF

END_FUNCTION_BLOCK
```
